(* IEC 61131-3 sources: Std_PalletMover/Class/MQTTClient_Interface (part 3) *)

      //-------------------------------
      //Logging
      //-------------------------------
      t_e_XML_Config::XC_Logging:

        if ProcessXML_ProcessConfig_Logging(pElement:=pThisElement) = FALSE then
          //CreateLog: Processing Logging Section of Configuration XML File Failed.

          Logging_InterfLog(usLevel     :=  MQTTCLIENTINTERFACE_LOGGING_LEVEL_ERR,
                            dMsgGroup   :=  MQCLIINF_LOG_ERROR_XML_CONFIG_LOGGING_NOT_OK_GRP,
                            dMsgNbr     :=  MQCLIINF_LOG_ERROR_XML_CONFIG_LOGGING_NOT_OK_MSG,
                            pMsg        :=  MQCLIINF_LOG_ERROR_XML_CONFIG_LOGGING_NOT_OK_TEXT,
                            pPara1      :=  NIL,
                            pPara2      :=  NIL,
                            pPara3      :=  NIL,
                            pPara4      :=  NIL);

          bOK := FALSE;
        end_if;

      //-------------------------------
      //Unknown, Skip
      //-------------------------------
      t_e_XML_Config::XC_Unknown:

    end_case;

    //Get the next client
    pThisElement := pThisElement^.pNext;

  end_while;

END_FUNCTION

FUNCTION MQTTClient_Interface::ProcessXML_ProcessConfig_GetElementType
	VAR_INPUT
		pElement 	: ^_XML_ELEMENT;
	END_VAR
	VAR_OUTPUT
		ElementType 	: t_e_XML_Config;
	END_VAR
  VAR
  	aString : ARRAY[0..MQTTCLIENT_INT_XML_CONFIG_MAX_LEN] of CHAR;
  END_VAR

  //Assume Unknown
  ElementType := XC_Unknown;

  if  pElement = NIL        |
      pElement^.Name = NIL  then
    return;
  end_if;

  //Convert the String to all upper for comparison to eliminate casing constraints
  SigCLib.StrNCpy(dst0  :=  #aString[0],
                  src0  :=  pElement^.Name,
                  count :=  MQTTCLIENT_INT_XML_CONFIG_MAX_LEN-1);

  aString[SigCLib.StrLen(str:=pElement^.Name)] := 0x00;

  SigCLib.StrUpr(ps1:=#aString[0]);

  if SigCLib.StrCmp(ps1:=#aString[0], ps2:=MQTTCLIENT_INT_XML_CONFIG_CLIENTID) = 0 then
    ElementType := XC_ClientID;
  elsif SigCLib.StrCmp(ps1:=#aString[0], ps2:=MQTTCLIENT_INT_XML_CONFIG_CONNECTION) = 0 then
    ElementType := XC_Connection;
  elsif SigCLib.StrCmp(ps1:=#aString[0], ps2:=MQTTCLIENT_INT_XML_CONFIG_RECONNECTION) = 0 then
    ElementType := XC_Reconnection;
  elsif SigCLib.StrCmp(ps1:=#aString[0], ps2:=MQTTCLIENT_INT_XML_CONFIG_TLS) = 0 then
    ElementType := XC_TLS;
  elsif SigCLib.StrCmp(ps1:=#aString[0], ps2:=MQTTCLIENT_INT_XML_CONFIG_LOGGING) = 0 then
    ElementType := XC_Logging;
  elsif SigCLib.StrCmp(ps1:=#aString[0], ps2:=MQTTCLIENT_INT_XML_CONFIG_WILL) = 0 then
    ElementType := XC_Will;
  end_if;

END_FUNCTION

FUNCTION MQTTClient_Interface::ProcessXML_ProcessConfig_ClientID
	VAR_INPUT
		pElement 	: ^_XML_ELEMENT;
	END_VAR
	VAR_OUTPUT
		bOK 	: BOOL;
	END_VAR

  //Assume Fail
  MQTTClientConfigData.Config.bClientIDSet := bOK := FALSE;

  //Get the ClientID from the XML File
  if  pElement                                                                              &
      pElement^.pText                                                                       &
      SigCLib.StrLen(str:=pElement^.pText) < sizeof(MQTTClientConfigData.Config.aClientID)  then

    SigCLib.MemSet( dst   :=  #MQTTClientConfigData.Config.aClientID[0],
                    c     :=  0x00,
                    len   :=  sizeof(MQTTClientConfigData.Config.aClientID));
    SigCLib.Utf8ToStr16(dst :=  #MQTTClientConfigData.Config.aClientID[0],
                        src :=  pElement^.pText);

    MQTTClientConfigData.Config.bClientIDSet := bOK := TRUE;

  end_if;

END_FUNCTION

FUNCTION MQTTClient_Interface::ProcessXML_GetElementType
	VAR_INPUT
		pElement 	: ^_XML_ELEMENT;
	END_VAR
	VAR_OUTPUT
		ElementType 	: t_e_XML;
	END_VAR
  VAR
  	aString : ARRAY[0..MTTCLIENT_INT_XML_CONFIG_DATAMAP_MAX_LEN] of CHAR;
  END_VAR

  //Assume Not Found
  ElementType := X_Unknown;

    //Convert the String to all upper for comparison to eliminate casing constraints
    SigCLib.StrNCpy(dst0  :=  #aString[0],
                    src0  :=  pElement^.Name,
                    count :=  MTTCLIENT_INT_XML_CONFIG_DATAMAP_MAX_LEN-1);

    aString[SigCLib.StrLen(str:=pElement^.Name)] := 0x00;

    SigCLib.StrUpr(ps1:=#aString[0]);

  if pElement then

    if SigCLib.StrCmp(ps1:=#aString[0], ps2:=MTTCLIENT_INT_XML_CONFIG_ELEMENT) = 0 then
      ElementType := X_Config;
      return;
    elsif SigCLib.StrCmp(ps1:=#aString[0], ps2:=MTTCLIENT_INT_XML_DATAMAP_ELEMENT) = 0 then
      ElementType := X_DataMap;
      return;
    end_if;

  end_if;

END_FUNCTION

FUNCTION MQTTClient_Interface::ProcessXML_ProcessDataMap
	VAR_INPUT
		pElement 	: ^_XML_ELEMENT;
	END_VAR
	VAR_OUTPUT
		bOK 	: BOOL;
	END_VAR
  VAR
  	pThisElement : ^_XML_ELEMENT;
  END_VAR

  //Assume Fail
  bOK := FALSE;

  if pElement = NIL then
    return;
  end_if;

  bOK := TRUE;
  pThisElement := pElement;

  //Step through all the children
  while pThisElement do

    //======================================================================
    //Based on the type of element, process
    //======================================================================
    case ProcessXML_ProcessDataMap_GetElementType(pElement:=pThisElement) of

      //-------------------------------
      //Unknown
      //-------------------------------
      t_e_XML_DataMap::XD_Unknown:

        //Create Log: Unexpected input in DataMap section

        Logging_InterfLog(usLevel     :=  MQTTCLIENTINTERFACE_LOGGING_LEVEL_ERR,
                          dMsgGroup   :=  MQCLIINF_LOG_ERROR_XML_DATAMAP_UNEXPECTED_ENTRY_GRP,
                          dMsgNbr     :=  MQCLIINF_LOG_ERROR_XML_DATAMAP_UNEXPECTED_ENTRY_MSG,
                          pMsg        :=  MQCLIINF_LOG_ERROR_XML_DATAMAP_UNEXPECTED_ENTRY_TEXT,
                          pPara1      :=  NIL,
                          pPara2      :=  NIL,
                          pPara3      :=  NIL,
                          pPara4      :=  NIL);

        bOK := FALSE;

      //-------------------------------
      //Topic Section
      //-------------------------------
      t_e_XML_DataMap::XD_TopicSection:

        if ProcessXML_ProcessDataMap_TopicSection(pElement:=pThisElement) = FALSE then

          bOK := FALSE;
          //Create Log: Failed Processing TopicSection in the DataMap Section

          Logging_InterfLog(usLevel     :=  MQTTCLIENTINTERFACE_LOGGING_LEVEL_ERR,
                            dMsgGroup   :=  MQCLIINF_LOG_ERROR_XML_DATAMAP_TOPICSECT_NOT_OK_GRP,
                            dMsgNbr     :=  MQCLIINF_LOG_ERROR_XML_DATAMAP_TOPICSECT_NOT_OK_MSG,
                            pMsg        :=  MQCLIINF_LOG_ERROR_XML_DATAMAP_TOPICSECT_NOT_OK_TEXT,
                            pPara1      :=  NIL,
                            pPara2      :=  NIL,
                            pPara3      :=  NIL,
                            pPara4      :=  NIL);
        end_if;

      //-------------------------------
      //Topic Endpoint
      //-------------------------------
      t_e_XML_DataMap::XD_TopicEndpoint:

        if ProcessXML_ProcessDataMap_TopicEndpoint(pElement:=pThisElement) = FALSE then
          bOK := FALSE;
          //Create Log: Failed Processing TopicEndpoint in the DataMap Section

          Logging_InterfLog(usLevel     :=  MQTTCLIENTINTERFACE_LOGGING_LEVEL_ERR,
                            dMsgGroup   :=  MQCLIINF_LOG_ERROR_XML_DATAMAP_TOPICENDPT_NOT_OK_GRP,
                            dMsgNbr     :=  MQCLIINF_LOG_ERROR_XML_DATAMAP_TOPICENDPT_NOT_OK_MSG,
                            pMsg        :=  MQCLIINF_LOG_ERROR_XML_DATAMAP_TOPICENDPT_NOT_OK_TEXT,
                            pPara1      :=  NIL,
                            pPara2      :=  NIL,
                            pPara3      :=  NIL,
                            pPara4      :=  NIL);

        end_if;

    end_case;

    pThisElement := pThisElement^.pNext;

  end_while;

END_FUNCTION

FUNCTION MQTTClient_Interface::ProcessXML_ProcessConfig_Connection
	VAR_INPUT
		pElement 	: ^_XML_ELEMENT;
	END_VAR
	VAR_OUTPUT
		bOK 	: BOOL;
	END_VAR
  VAR
    pThisElement : ^_XML_ELEMENT;
    aString : ARRAY[0..MQTTCLIENT_INT_XML_CONFIG_CONN_MAX_LEN] of CHAR;
  END_VAR

  bOK := FALSE;

  //Process the Connect Config
  if pElement             &
     pElement^.pChildren  then

    //==========================================================
    //Set Parameters
    //==========================================================
    pThisElement := pElement^.pChildren;

    while pThisElement        &
          pThisElement^.Name  &
          pThisElement^.pText do

      //Convert the String to all upper for comparison to eliminate casing constraints
      SigCLib.StrNCpy(dst0  :=  #aString[0],
                      src0  :=  pThisElement^.Name,
                      count :=  MQTTCLIENT_INT_XML_CONFIG_CONN_MAX_LEN-1);

      aString[SigCLib.StrLen(str:=pThisElement^.Name)] := 0x00;

      SigCLib.StrUpr(ps1:=#aString[0]);

      //------------------------------------------------------------------------------------------------------
      //Hostname
      //------------------------------------------------------------------------------------------------------
      if SigCLib.StrCmp(ps1:=#aString[0], ps2:=MQTTCLIENT_INT_XML_CONFIG_CONN_HOSTNAME) = 0 then

        if SigCLib.StrLen(str:=pThisElement^.pText) < MQTTCLIENT_HOSTNAME_MAX_LEN then
          SigCLib.Utf8ToStr16(dst:=#MQTTClientConfigData.Config.Connect.aHostname[0], src:=pThisElement^.pText);
          MQTTClientConfigData.Config.Connect.ValuesSet.Hostname := TRUE;
        end_if;

      //------------------------------------------------------------------------------------------------------
      //Port
      //------------------------------------------------------------------------------------------------------
      elsif SigCLib.StrCmp(ps1:=#aString[0], ps2:=MQTTCLIENT_INT_XML_CONFIG_CONN_PORT) = 0 then

        if SigCLib.StrLen(str:=pThisElement^.pText) < MQTTCLIENTINTERFACE_CONNECT_PORT_MAX_LEN then
          MQTTClientConfigData.Config.Connect.iPort := to_int(SigCLib.AToI(ps1:=pThisElement^.pText));
          MQTTClientConfigData.Config.Connect.ValuesSet.Port := TRUE;
        end_if;

      //------------------------------------------------------------------------------------------------------
      //Keepalive
      //------------------------------------------------------------------------------------------------------
      elsif SigCLib.StrCmp(ps1:=#aString[0], ps2:=MQTTCLIENT_INT_XML_CONFIG_CONN_KEEPALIVE) = 0 then

        if SigCLib.StrLen(str:=pThisElement^.pText) < MQTTCLIENTINTERFACE_CONNECT_KEEPALIVE_MAX_LEN then
          MQTTClientConfigData.Config.Connect.iKeepalive := to_int(SigCLib.AToI(ps1:=pThisElement^.pText));
          MQTTClientConfigData.Config.Connect.ValuesSet.Keepalive := TRUE;
        end_if;

      //------------------------------------------------------------------------------------------------------
      //Max Inflight
      //------------------------------------------------------------------------------------------------------
      elsif SigCLib.StrCmp(ps1:=#aString[0], ps2:=MQTTCLIENT_INT_XML_CONFIG_CONN_MAXINFLIGHT) = 0 then

        if SigCLib.StrLen(str:=pThisElement^.pText) < MQTTCLIENTINTERFACE_CONNECT_INFLIGHT_MAX_LEN then
          MQTTClientConfigData.Config.Connect.iMaxInflightMessages := to_int(SigCLib.AToI(ps1:=pThisElement^.pText));
          MQTTClientConfigData.Config.Connect.ValuesSet.MaxInflight := TRUE;
        end_if;

      //------------------------------------------------------------------------------------------------------
      //Username
      //------------------------------------------------------------------------------------------------------
      elsif SigCLib.StrCmp(ps1:=#aString[0], ps2:=MQTTCLIENT_INT_XML_CONFIG_CONN_USERNAME) = 0 then

        if SigCLib.StrLen(str:=pThisElement^.pText) < MQTTCLIENTINTERFACE_CONNECT_USERNAME_MAX_LEN then
          SigCLib.Utf8ToStr16(dst:=#MQTTClientConfigData.Config.Connect.aUsername[0], src:=pThisElement^.pText);
          MQTTClientConfigData.Config.Connect.ValuesSet.Username := TRUE;
        end_if;

      //------------------------------------------------------------------------------------------------------
      //Password
      //------------------------------------------------------------------------------------------------------
      elsif SigCLib.StrCmp(ps1:=#aString[0], ps2:=MQTTCLIENT_INT_XML_CONFIG_CONN_PASSWORD) = 0 then

        if SigCLib.StrLen(str:=pThisElement^.pText) < MQTTCLIENTINTERFACE_CONNECT_PASSWORD_MAX_LEN then
          SigCLib.Utf8ToStr16(dst:=#MQTTClientConfigData.Config.Connect.aPassword[0], src:=pThisElement^.pText);
          MQTTClientConfigData.Config.Connect.ValuesSet.Password := TRUE;
        end_if;

      end_if;

      pThisElement := pThisElement^.pNext;

    end_while;

    //Return is OK if atleast the Hostname is set
    bOK := MQTTClientConfigData.Config.Connect.ValuesSet.Hostname;

  end_if;

END_FUNCTION

FUNCTION MQTTClient_Interface::ProcessXML_ProcessConfig_Will
	VAR_INPUT
		pElement 	: ^_XML_ELEMENT;
	END_VAR
	VAR_OUTPUT
		bOK 	: BOOL;
	END_VAR
  VAR
    pThisElement : ^_XML_ELEMENT;
  	aString : ARRAY[0..MQTTCLIENT_INT_XML_CONFIG_WILL_MAX_LEN] of CHAR;
  END_VAR

  bOK := FALSE;

  //Process the Connect Config
  if pElement             &
     pElement^.pChildren  then

    //==========================================================
    //Set Parameters
    //==========================================================
    pThisElement := pElement^.pChildren;

    while pThisElement        &
          pThisElement^.Name  &
          pThisElement^.pText do

      //Convert the String to all upper for comparison to eliminate casing constraints
      SigCLib.StrNCpy(dst0  :=  #aString[0],
                      src0  :=  pThisElement^.Name,
                      count :=  MQTTCLIENT_INT_XML_CONFIG_WILL_MAX_LEN-1);

      aString[SigCLib.StrLen(str:=pThisElement^.Name)] := 0x00;

      SigCLib.StrUpr(ps1:=#aString[0]);

      //------------------------------------------------------------------------------------------------------
      //Topic
      //------------------------------------------------------------------------------------------------------
      if SigCLib.StrCmp(ps1:=#aString[0], ps2:=MQTTCLIENT_INT_XML_CONFIG_WILL_TOPIC) = 0 then

        if SigCLib.StrLen(str:=pThisElement^.pText) < MQTTCLIENTINTERFACE_WILL_TOPIC_MAX_LEN then
          SigCLib.Utf8ToStr16(dst:=#MQTTClientConfigData.Config.Will.aTopic[0], src:=pThisElement^.pText);
          MQTTClientConfigData.Config.Will.ValuesSet.Topic := TRUE;
        end_if;

      //------------------------------------------------------------------------------------------------------
      //Payload
      //------------------------------------------------------------------------------------------------------
      elsif SigCLib.StrCmp(ps1:=#aString[0], ps2:=MQTTCLIENT_INT_XML_CONFIG_WILL_PLTEXT) = 0 then

        if SigCLib.StrLen(str:=pThisElement^.pText) < MQTTCLIENTINTERFACE_WILL_PAYLOAD_MAX_LEN then
          //Data from XML Structure must be text, although the payload in the MQTT Client allows for Non-UTF8 input
          SigCLib.StrCpy(dst0:=#MQTTClientConfigData.Config.Will.aPayload[0], src0:=pThisElement^.pText);
          MQTTClientConfigData.Config.Will.ValuesSet.Payload := TRUE;
        end_if;

      //------------------------------------------------------------------------------------------------------
      //QoS
      //------------------------------------------------------------------------------------------------------
      elsif SigCLib.StrCmp(ps1:=#aString[0], ps2:=MQTTCLIENT_INT_XML_CONFIG_WILL_QOS) = 0 then

        if SigCLib.StrLen(str:=pThisElement^.pText) = MQTTCLIENTINTERFACE_WILL_QOS_MAX_LEN then

          MQTTClientConfigData.Config.Will.ValuesSet.QoS := TRUE;

          //=======================================
          //Conv QoS CHAR to INT
          //=======================================
          case pThisElement^.pText^ of
            //-----------------------------------
            //QoS 0
            //-----------------------------------
            MQTTCLIENT_INT_XML_CONFIG_WILL_QOS_0:

              MQTTClientConfigData.Config.Will.iQoS := 0;

            //-----------------------------------
            //QoS 1
            //-----------------------------------
            MQTTCLIENT_INT_XML_CONFIG_WILL_QOS_1:

              MQTTClientConfigData.Config.Will.iQoS := 1;

            //-----------------------------------
            //QoS 2
            //-----------------------------------
            MQTTCLIENT_INT_XML_CONFIG_WILL_QOS_2:

              MQTTClientConfigData.Config.Will.iQoS := 2;

          //Not a valid Character
          else

            MQTTClientConfigData.Config.Will.ValuesSet.QoS := FALSE;

          end_case;

        end_if;

      //------------------------------------------------------------------------------------------------------
      //Retain
      //------------------------------------------------------------------------------------------------------
      elsif SigCLib.StrCmp(ps1:=#aString[0], ps2:=MQTTCLIENT_INT_XML_CONFIG_WILL_RETAIN) = 0 then

        if SigCLib.StrLen(str:=pThisElement^.pText) = MQTTCLIENT_INT_XML_CONFIG_WILL_RETAIN_MAXLEN then

          //===========================
          //Set Log based on text value
          //===========================
          case pThisElement^.pText^ of
            //---------------------------------
            //True
            //---------------------------------
            MQTTCLIENT_INT_XML_CONFIG_WILL_RETAIN_TRUE:
              MQTTClientConfigData.Config.Will.bRetain := TRUE;
              MQTTClientConfigData.Config.Will.ValuesSet.RetainWill := TRUE;
            //---------------------------------
            //False
            //---------------------------------
            MQTTCLIENT_INT_XML_CONFIG_WILL_RETAIN_FALSE:
              MQTTClientConfigData.Config.Will.bRetain := FALSE;
              MQTTClientConfigData.Config.Will.ValuesSet.RetainWill := TRUE;
          end_case;

        end_if;

      end_if;

      pThisElement := pThisElement^.pNext;

    end_while;

    //All Paras are required
    bOK :=  MQTTClientConfigData.Config.Will.ValuesSet.Topic      &
            MQTTClientConfigData.Config.Will.ValuesSet.Payload    &
            MQTTClientConfigData.Config.Will.ValuesSet.QoS        &
            MQTTClientConfigData.Config.Will.ValuesSet.RetainWill;

  end_if;

END_FUNCTION

FUNCTION MQTTClient_Interface::ProcessXML_ProcessConfig_Reconnection
	VAR_INPUT
		pElement 	: ^_XML_ELEMENT;
	END_VAR
	VAR_OUTPUT
		bOK 	: BOOL;
	END_VAR
  VAR
    pThisElement : ^_XML_ELEMENT;
    aString : ARRAY[0..MQTTCLIENT_INT_XML_CONFIG_RECONN_MAXLEN] of CHAR;
  END_VAR

  bOK := FALSE;

  //Process the Connect Config
  if pElement             &
     pElement^.pChildren  then

    //==========================================================
    //Set Parameters
    //==========================================================
    pThisElement := pElement^.pChildren;

    while pThisElement        &
          pThisElement^.Name  &
          pThisElement^.pText do

      //Convert the String to all upper for comparison to eliminate casing constraints
      SigCLib.StrNCpy(dst0  :=  #aString[0],
                      src0  :=  pThisElement^.Name,
                      count :=  MQTTCLIENT_INT_XML_CONFIG_RECONN_MAXLEN-1);

      aString[SigCLib.StrLen(str:=pThisElement^.Name)] := 0x00;

      SigCLib.StrUpr(ps1:=#aString[0]);

      //------------------------------------------------------------------------------------------------------
      //Min Interval
      //------------------------------------------------------------------------------------------------------
      if SigCLib.StrCmp(ps1:=#aString[0], ps2:=MQTTCLIENT_INT_XML_CONFIG_RECONN_MININT) = 0 then

        if SigCLib.StrLen(str:=pThisElement^.pText) < MQTTCLIENTINTERFACE_RECONNECT_MININT_MAX_LEN then
          MQTTClientConfigData.Config.Reconnect.iMinInterval := to_int(SigCLib.AToI(ps1:=pThisElement^.pText));
          MQTTClientConfigData.Config.Reconnect.ValuesSet.MinInterval := TRUE;
        end_if;

      //------------------------------------------------------------------------------------------------------
      //Max Interval
      //------------------------------------------------------------------------------------------------------
      elsif SigCLib.StrCmp(ps1:=#aString[0], ps2:=MQTTCLIENT_INT_XML_CONFIG_RECONN_MAXINT) = 0 then

        if SigCLib.StrLen(str:=pThisElement^.pText) < MQTTCLIENTINTERFACE_RECONNECT_MAXINT_MAX_LEN then
          MQTTClientConfigData.Config.Reconnect.iMaxInterval := to_int(SigCLib.AToI(ps1:=pThisElement^.pText));
          MQTTClientConfigData.Config.Reconnect.ValuesSet.MaxInterval := TRUE;
        end_if;

      //------------------------------------------------------------------------------------------------------
      //Exponential Scale
      //------------------------------------------------------------------------------------------------------
      elsif SigCLib.StrCmp(ps1:=#aString[0], ps2:=MQTTCLIENT_INT_XML_CONFIG_RECONN_EXPSCALE) = 0 then

        if SigCLib.StrLen(str:=pThisElement^.pText) = SigCLib.StrLen(str:=MQTTCLIENT_INT_XML_CONFIG_RECONNECT_EXP_ON) then
          MQTTClientConfigData.Config.Reconnect.bExponential := (SigCLib.StrCmp(ps1:=pThisElement^.pText, ps2:=MQTTCLIENT_INT_XML_CONFIG_RECONNECT_EXP_ON) = 0);
          MQTTClientConfigData.Config.Reconnect.ValuesSet.ExponentialScale := TRUE;
        end_if;

      end_if;

      pThisElement := pThisElement^.pNext;

    end_while;

    //Return is OK if all is set
    bOK :=  MQTTClientConfigData.Config.Reconnect.ValuesSet.MinInterval &
            MQTTClientConfigData.Config.Reconnect.ValuesSet.MaxInterval &
            MQTTClientConfigData.Config.Reconnect.ValuesSet.ExponentialScale;

  end_if;

END_FUNCTION

FUNCTION MQTTClient_Interface::ProcessXML_ProcessConfig_TLS
	VAR_INPUT
		pElement 	: ^_XML_ELEMENT;
	END_VAR
	VAR_OUTPUT
		bOK 	: BOOL;
	END_VAR
  VAR
    pThisElement : ^_XML_ELEMENT;
    aString : ARRAY[0..MQTTCLIENT_INT_XML_CONFIG_TLS_MAXLEN] of CHAR;
  END_VAR

  bOK := FALSE;

  //Process the Connect Config
  if pElement             &
     pElement^.pChildren  then

    MQTTClientConfigData.Config.TLS.ValuesSet.TLS := TRUE;

    //==========================================================
    //Set Parameters
    //==========================================================
    pThisElement := pElement^.pChildren;

    while pThisElement        &
          pThisElement^.Name  &
          pThisElement^.pText do

      //Convert the String to all upper for comparison to eliminate casing constraints
      SigCLib.StrNCpy(dst0  :=  #aString[0],
                      src0  :=  pThisElement^.Name,
                      count :=  MQTTCLIENT_INT_XML_CONFIG_TLS_MAXLEN-1);

      aString[SigCLib.StrLen(str:=pThisElement^.Name)] := 0x00;

      SigCLib.StrUpr(ps1:=#aString[0]);

      //------------------------------------------------------------------------------------------------------
      //cafile
      //------------------------------------------------------------------------------------------------------
      if SigCLib.StrCmp(ps1:=#aString[0], ps2:=MQTTCLIENT_INT_XML_CONFIG_TLS_CAFILE) = 0 then

        if SigCLib.StrLen(str:=pThisElement^.pText) < MQTTCLIENTINTERFACE_TLS_CAFILE_MAX_LEN then
          SigCLib.StrCpy(dst0:=#MQTTClientConfigData.Config.TLS.aCAFile[0], src0:=pThisElement^.pText);
          MQTTClientConfigData.Config.TLS.ValuesSet.CAFile := TRUE;
        end_if;

      //------------------------------------------------------------------------------------------------------
      //certfile
      //------------------------------------------------------------------------------------------------------
      elsif SigCLib.StrCmp(ps1:=#aString[0], ps2:=MQTTCLIENT_INT_XML_CONFIG_TLS_CERTFILE) = 0 then

        if SigCLib.StrLen(str:=pThisElement^.pText) < MQTTCLIENTINTERFACE_TLS_CERTFILE_MAX_LEN then
          SigCLib.StrCpy(dst0:=#MQTTClientConfigData.Config.TLS.aCertFile[0], src0:=pThisElement^.pText);
          MQTTClientConfigData.Config.TLS.ValuesSet.CertFile := TRUE;
        end_if;

      //------------------------------------------------------------------------------------------------------
      //keyfile
      //------------------------------------------------------------------------------------------------------
      elsif SigCLib.StrCmp(ps1:=#aString[0], ps2:=MQTTCLIENT_INT_XML_CONFIG_TLS_KEYFILE) = 0 then

        if SigCLib.StrLen(str:=pThisElement^.pText) < MQTTCLIENTINTERFACE_TLS_KEYFILE_MAX_LEN then
          SigCLib.StrCpy(dst0:=#MQTTClientConfigData.Config.TLS.aKeyFile[0], src0:=pThisElement^.pText);
          MQTTClientConfigData.Config.TLS.ValuesSet.KeyFile := TRUE;
        end_if;

      //------------------------------------------------------------------------------------------------------
      //pw
      //------------------------------------------------------------------------------------------------------
      elsif SigCLib.StrCmp(ps1:=#aString[0], ps2:=MQTTCLIENT_INT_XML_CONFIG_TLS_PW) = 0 then

        if SigCLib.StrLen(str:=pThisElement^.pText) < MQTTCLIENTINTERFACE_TLS_PASSWORD_MAX_LEN then
          SigCLib.StrCpy(dst0:=#MQTTClientConfigData.Config.TLS.aPassword[0], src0:=pThisElement^.pText);
          MQTTClientConfigData.Config.TLS.ValuesSet.Password := TRUE;
        end_if;

      end_if;

      pThisElement := pThisElement^.pNext;

    end_while;

    //No input is required
    bOK := TRUE;

  end_if;

END_FUNCTION

FUNCTION MQTTClient_Interface::ProcessXML_ProcessConfig_Logging
	VAR_INPUT
		pElement 	: ^_XML_ELEMENT;
	END_VAR
	VAR_OUTPUT
		bOK 	: BOOL;
	END_VAR
  VAR
    pThisElement : ^_XML_ELEMENT;
    aString : ARRAY[0..MQTTCLIENT_INT_XML_CONFIG_LOG_MAX_LEN] of CHAR;
  END_VAR

  bOK := FALSE;

  MQTTClientConfigData.Config.Logging.bLogSet       := FALSE;
  MQTTClientConfigData.Config.Logging.bdActiveLogs  := 0;

  //Process the Logging Config
  if pElement             &
     pElement^.pChildren  then

    //==========================================================
    //Set Parameters
    //==========================================================
    pThisElement := pElement^.pChildren;

    while pThisElement        &
          pThisElement^.Name  &
          pThisElement^.pText do

      //Convert the String to all upper for comparison to eliminate casing constraints
      SigCLib.StrNCpy(dst0  :=  #aString[0],
                      src0  :=  pThisElement^.Name,
                      count :=  MQTTCLIENT_INT_XML_CONFIG_LOG_MAX_LEN-1);

      aString[SigCLib.StrLen(str:=pThisElement^.Name)] := 0x00;

      SigCLib.StrUpr(ps1:=#aString[0]);

      //If any log entry is present, set the ValuePresent
      MQTTClientConfigData.Config.Logging.bLogSet := TRUE;

      //------------------------------------------------------------------------------------------------------
      //Info
      //------------------------------------------------------------------------------------------------------
      if SigCLib.StrCmp(ps1:=#aString[0], ps2:=MQTTCLIENT_INT_XML_CONFIG_LOG_INFO) = 0 then

        if SigCLib.StrLen(str:=pThisElement^.pText) = MQTTCLIENTINTERFACE_LOG_ON_OFF_MAX_LEN then

          //===========================
          //Set Log based on text value
          //===========================
          case pThisElement^.pText^ of
            //---------------------------------
            //Off
            //---------------------------------
            MQTTCLIENT_INT_XML_CONFIG_LOG_OFF:
              MQTTClientConfigData.Config.Logging.bdActiveLogs$BDINT := MQTTClientConfigData.Config.Logging.bdActiveLogs$BDINT AND (NOT (MQTTCLIENTINTERFACE_LOGGING_LEVEL_INFO$BDINT));
            //---------------------------------
            //On
            //---------------------------------
            MQTTCLIENT_INT_XML_CONFIG_LOG_ON:
              MQTTClientConfigData.Config.Logging.bdActiveLogs$BDINT := MQTTClientConfigData.Config.Logging.bdActiveLogs$BDINT OR MQTTCLIENTINTERFACE_LOGGING_LEVEL_INFO$BDINT;
          end_case;

        end_if;

      //------------------------------------------------------------------------------------------------------
      //Notice
      //------------------------------------------------------------------------------------------------------
      elsif SigCLib.StrCmp(ps1:=#aString[0], ps2:=MQTTCLIENT_INT_XML_CONFIG_LOG_NOTICE) = 0 then

        if SigCLib.StrLen(str:=pThisElement^.pText) = MQTTCLIENTINTERFACE_LOG_ON_OFF_MAX_LEN then

          //===========================
          //Set Log based on text value
          //===========================
          case pThisElement^.pText^ of
            //---------------------------------
            //Off
            //---------------------------------
            MQTTCLIENT_INT_XML_CONFIG_LOG_OFF:
              MQTTClientConfigData.Config.Logging.bdActiveLogs$BDINT := MQTTClientConfigData.Config.Logging.bdActiveLogs$BDINT AND (NOT (MQTTCLIENTINTERFACE_LOGGING_LEVEL_NOTICE$BDINT));
            //---------------------------------
            //On
            //---------------------------------
            MQTTCLIENT_INT_XML_CONFIG_LOG_ON:
              MQTTClientConfigData.Config.Logging.bdActiveLogs := MQTTClientConfigData.Config.Logging.bdActiveLogs OR MQTTCLIENTINTERFACE_LOGGING_LEVEL_NOTICE$BDINT;
          end_case;

        end_if;

      //------------------------------------------------------------------------------------------------------
      //Warning
      //------------------------------------------------------------------------------------------------------
      elsif SigCLib.StrCmp(ps1:=#aString[0], ps2:=MQTTCLIENT_INT_XML_CONFIG_LOG_WARNING) = 0 then

        if SigCLib.StrLen(str:=pThisElement^.pText) = MQTTCLIENTINTERFACE_LOG_ON_OFF_MAX_LEN then

          //===========================
          //Set Log based on text value
          //===========================
          case pThisElement^.pText^ of
            //---------------------------------
            //Off
            //---------------------------------
            MQTTCLIENT_INT_XML_CONFIG_LOG_OFF:
              MQTTClientConfigData.Config.Logging.bdActiveLogs$BDINT := MQTTClientConfigData.Config.Logging.bdActiveLogs$BDINT AND (NOT MQTTCLIENTINTERFACE_LOGGING_LEVEL_WARNING);
            //---------------------------------
            //On
            //---------------------------------
            MQTTCLIENT_INT_XML_CONFIG_LOG_ON:
              MQTTClientConfigData.Config.Logging.bdActiveLogs := MQTTClientConfigData.Config.Logging.bdActiveLogs OR MQTTCLIENTINTERFACE_LOGGING_LEVEL_WARNING$BDINT;
          end_case;

        end_if;

      //------------------------------------------------------------------------------------------------------
      //Error
      //------------------------------------------------------------------------------------------------------
      elsif SigCLib.StrCmp(ps1:=#aString[0], ps2:=MQTTCLIENT_INT_XML_CONFIG_LOG_ERROR) = 0 then

        if SigCLib.StrLen(str:=pThisElement^.pText) = MQTTCLIENTINTERFACE_LOG_ON_OFF_MAX_LEN then

          //===========================
          //Set Log based on text value
          //===========================
          case pThisElement^.pText^ of
            //---------------------------------
            //Off
            //---------------------------------
            MQTTCLIENT_INT_XML_CONFIG_LOG_OFF:
              MQTTClientConfigData.Config.Logging.bdActiveLogs$BDINT := MQTTClientConfigData.Config.Logging.bdActiveLogs$BDINT AND (NOT (MQTTCLIENTINTERFACE_LOGGING_LEVEL_ERR$BDINT));
            //---------------------------------
            //On
            //---------------------------------
            MQTTCLIENT_INT_XML_CONFIG_LOG_ON:
              MQTTClientConfigData.Config.Logging.bdActiveLogs$BDINT := MQTTClientConfigData.Config.Logging.bdActiveLogs$BDINT OR MQTTCLIENTINTERFACE_LOGGING_LEVEL_ERR$BDINT;
          end_case;

        end_if;

      //------------------------------------------------------------------------------------------------------
      //Debugging
      //------------------------------------------------------------------------------------------------------
      elsif SigCLib.StrCmp(ps1:=#aString[0], ps2:=MQTTCLIENT_INT_XML_CONFIG_LOG_DEBUGGING) = 0 then

        if SigCLib.StrLen(str:=pThisElement^.pText) = MQTTCLIENTINTERFACE_LOG_ON_OFF_MAX_LEN then

          //===========================
          //Set Log based on text value
          //===========================
          case pThisElement^.pText^ of
            //---------------------------------
            //Off
            //---------------------------------
            MQTTCLIENT_INT_XML_CONFIG_LOG_OFF:
              MQTTClientConfigData.Config.Logging.bdActiveLogs$BDINT := MQTTClientConfigData.Config.Logging.bdActiveLogs$BDINT AND (NOT (MQTTCLIENTINTERFACE_LOGGING_LEVEL_DEBUG$BDINT));
            //---------------------------------
            //On
            //---------------------------------
            MQTTCLIENT_INT_XML_CONFIG_LOG_ON:
              MQTTClientConfigData.Config.Logging.bdActiveLogs$BDINT := MQTTClientConfigData.Config.Logging.bdActiveLogs$BDINT OR MQTTCLIENTINTERFACE_LOGGING_LEVEL_DEBUG$BDINT;
          end_case;

        end_if;

      end_if;

      pThisElement := pThisElement^.pNext;

    end_while;

    //Return is always OK
    bOK := TRUE;

  end_if;

END_FUNCTION

FUNCTION MQTTClient_Interface::ProcessXML_ProcessDataMap_GetElementType
	VAR_INPUT
		pElement 	: ^_XML_ELEMENT;
	END_VAR
	VAR_OUTPUT
		ElementType 	: t_e_XML_DataMap;
	END_VAR
  VAR
  	aString : ARRAY[0..MQTTCLIENT_INT_XML_DATAMAP_TOPIC_SECT_END_MAX_LEN] of CHAR;
  END_VAR

  //Assume Unknown
  ElementType := XD_Unknown;

  if pElement then

  //Convert the String to all upper for comparison to eliminate casing constraints
    SigCLib.StrNCpy(dst0  :=  #aString[0],
                    src0  :=  pElement^.Name,
                    count :=  MQTTCLIENT_INT_XML_DATAMAP_TOPIC_SECT_END_MAX_LEN-1);

    aString[SigCLib.StrLen(str:=pElement^.Name)] := 0x00;

    SigCLib.StrUpr(ps1:=#aString[0]);

    if SigCLib.StrCmp(ps1:=#aString[0], ps2:=MQTTCLIENT_INT_XML_DATAMAP_TOPICSECTION) = 0 then
      ElementType := XD_TopicSection;
    elsif SigCLib.StrCmp(ps1:=#aString[0], ps2:=MQTTCLIENT_INT_XML_DATAMAP_TOPICENDPOINT) = 0 then
      ElementType := XD_TopicEndpoint;
    end_if;

  end_if;

END_FUNCTION

FUNCTION MQTTClient_Interface::ProcessXML_ProcessDataMap_TopicSection
	VAR_INPUT
		pElement 	: ^_XML_ELEMENT;
	END_VAR
	VAR_OUTPUT
		bOK 	: BOOL;
	END_VAR
  VAR
  	pChild : ^_XML_ELEMENT;
    tmpPara : DINT;
  	aString : ARRAY[0..MQTTCLIENT_INT_XML_DATAMAP_TOPICSECTION_ATTR_MAX_LEN] of CHAR;
  END_VAR

  //Assume Fail
  bOK := FALSE;

  if pElement = NIL                           |
     pElement^.Attributes.pList = NIL         |
     pElement^.Attributes.pList^.Name = NIL   |
     pElement^.Attributes.pList^.Value = NIL then
    return;
  end_if;

  //Convert the String to all upper for comparison to eliminate casing constraints
    SigCLib.StrNCpy(dst0  :=  #aString[0],
                    src0  :=  pElement^.Attributes.pList^.Name,
                    count :=  MQTTCLIENT_INT_XML_DATAMAP_TOPICSECTION_ATTR_MAX_LEN-1);

    aString[SigCLib.StrLen(str:=pElement^.Attributes.pList^.Name)] := 0x00;

    SigCLib.StrUpr(ps1:=#aString[0]);

  //Append the section to the Topicname being built (First and only Attribute should be "name")
  if SigCLib.StrCmp(ps1:=#aString[0], ps2:=MQTTCLIENT_INT_XML_DATAMAP_TOPICSECTION_ATTR_NAME) = 0 then

    //Topic Depth OK
    if Config.pDataMapConfig^.udTopicStringDepth >= 0 &
       Config.pDataMapConfig^.udTopicStringDepth <  MQTTCLIENT_INT_XML_DATAMAP_TOPICSECTION_MAXSECDEPTH then

      //Value set but too long
      if  (SigCLib.StrLen(str:=pElement^.Attributes.pList^.Value) >= MQTTCLIENT_INT_XML_DATAMAP_TOPICSECTION_MAXSECLEN) then

        //Create Log: DataMap, Processing topic Section failed - Section title too long

        Logging_InterfLog(usLevel     :=  MQTTCLIENTINTERFACE_LOGGING_LEVEL_ERR,
                          dMsgGroup   :=  MQCLIINF_LOG_ERROR_XML_DATAMAP_TS_TITLE_LEN_GRP,
                          dMsgNbr     :=  MQCLIINF_LOG_ERROR_XML_DATAMAP_TS_TITLE_LEN_MSG,
                          pMsg        :=  MQCLIINF_LOG_ERROR_XML_DATAMAP_TS_TITLE_LEN_TEXT,
                          pPara1      :=  NIL,
                          pPara2      :=  NIL,
                          pPara3      :=  NIL,
                          pPara4      :=  NIL);

        return;

      //Value not set
      elsif pElement^.Attributes.pList^.Value = NIL then

        //Create Log: DataMap, Processing topic Section failed - Section title empty

        Logging_InterfLog(usLevel     :=  MQTTCLIENTINTERFACE_LOGGING_LEVEL_ERR,
                          dMsgGroup   :=  MQCLIINF_LOG_ERROR_XML_DATAMAP_TS_TITLE_EMPTY_GRP,
                          dMsgNbr     :=  MQCLIINF_LOG_ERROR_XML_DATAMAP_TS_TITLE_EMPTY_MSG,
                          pMsg        :=  MQCLIINF_LOG_ERROR_XML_DATAMAP_TS_TITLE_EMPTY_TEXT,
                          pPara1      :=  NIL,
                          pPara2      :=  NIL,
                          pPara3      :=  NIL,
                          pPara4      :=  NIL);

        return;

      //Value set and OK
      else

        SigCLib.MemSet( dst :=  #Config.pDataMapConfig^.aTopicStrings[Config.pDataMapConfig^.udTopicStringDepth][0],
                        c   :=  0x00,
                        len :=  sizeof(t_s_TopicString));
        SigCLib.StrCpy( dst0  :=  #Config.pDataMapConfig^.aTopicStrings[Config.pDataMapConfig^.udTopicStringDepth][0],
                        src0  :=  pElement^.Attributes.pList^.Value);
        Config.pDataMapConfig^.udTopicStringDepth += 1;
        bOK := TRUE;

      end_if;

    //Exceeded maximum topic depth
    elsif Config.pDataMapConfig^.udTopicStringDepth >= MQTTCLIENT_INT_XML_DATAMAP_TOPICSECTION_MAXSECDEPTH then

      //Create Log: DataMap, Processing topic section failed, maximum topic depth exceeded.

      tmpPara := MQTTCLIENT_INT_XML_DATAMAP_TOPICSECTION_MAXSECDEPTH;

      Logging_InterfLog(usLevel     :=  MQTTCLIENTINTERFACE_LOGGING_LEVEL_ERR,
                        dMsgGroup   :=  MQCLIINF_LOG_ERROR_XML_DATAMAP_TS_MAX_DEPTH_EXCEED_GRP,
                        dMsgNbr     :=  MQCLIINF_LOG_ERROR_XML_DATAMAP_TS_MAX_DEPTH_EXCEED_MSG,
                        pMsg        :=  MQCLIINF_LOG_ERROR_XML_DATAMAP_TS_MAX_DEPTH_EXCEED_TEXT,
                        pPara1      :=  #Config.pDataMapConfig^.udTopicStringDepth$DINT,
                        pPara2      :=  #tmpPara,
                        pPara3      :=  NIL,
                        pPara4      :=  NIL);

    end_if;

    //Process any children the Section has
    pChild := pElement^.pChildren;
    if pChild then
      bOK := ProcessXML_ProcessDataMap(pElement:=pChild);
    else
      bOK := FALSE;
    end_if;

    if Config.pDataMapConfig^.udTopicStringDepth >= 1 then
      Config.pDataMapConfig^.udTopicStringDepth -= 1;
    end_if;

  end_if;

END_FUNCTION

FUNCTION MQTTClient_Interface::ProcessXML_ProcessDataMap_TopicEndpoint
	VAR_INPUT
		pElement 	: ^_XML_ELEMENT;
	END_VAR
	VAR_OUTPUT
		bOK 	: BOOL;
	END_VAR
  VAR
    aTopicString    : ARRAY[0..MQTTCLIENT_TOPIC_MAX_LEN] of CHAR;
  	udAtt, udCount  : UDINT;
    pAtt            : ^_XML_ATTRIBUTE;
    aEndpointName   : ARRAY[0..MQTTCLIENT_INT_XML_DATAMAP_TOPICENDPOINT_NAME_MAX_LEN] of CHAR;
    aElement        : ARRAY[0..MQTTCLIENT_INT_XML_DATAMAP_TOPICENDPOINT_ELEMENT_MAX_LEN] of CHAR;
    Operation       : t_e_DataMap_Operations;
    udInterval      : UDINT;
    DataType        : t_e_DataMap_DataTypes;
    bNameSet, bElementSet : BOOL;
    udLen           : UDINT;
    iQoS            : INT;
    DRSRetain       : t_e_DataMap_RetainStates;
    DataMapRet      : t_e_DataMap_RetCode;
    tmpPara         : DINT;
    aString         : ARRAY[0..MQTTCLIENT_INT_XML_DATAMAP_TOPICENDPOINT_ATTR_MAX_LEN] of CHAR;
  END_VAR

  //Assume Fail
  bOK := FALSE;

  if pElement = NIL                                                                 |
     pElement^.Attributes.no = 0                                                    |
     pElement^.Attributes.no > MQTTCLIENT_INT_XML_DATAMAP_TOPICENDPOINT_MAX_ATTRS   |
     pElement^.Attributes.pList = NIL                                               then
    return;
  end_if;

  //Set Default Values
  Operation   := DO_Subscribe;
  udInterval  := 0;
  DataType    := DD_DINT;
  bNameSet    := bElementSet := FALSE;
  iQoS        := 0;
  DRSRetain   := DRS_False;

  udAtt := pElement^.Attributes.no;

  while udAtt > 0 do

    //=======================
    //Process the Attribute
    //=======================
    pAtt := ((pElement^.Attributes.pList$UDINT) + (udAtt-1)*sizeof(_XML_ATTRIBUTE))$^_XML_ATTRIBUTE;

    if pAtt^.Name = NIL |
       pAtt^.Value = NIL then
      return;
    end_if;

    //Convert the String to all upper for comparison to eliminate casing constraints
    SigCLib.StrNCpy(dst0  :=  #aString[0],
                    src0  :=  pAtt^.Name$^CHAR,
                    count :=  MQTTCLIENT_INT_XML_DATAMAP_TOPICENDPOINT_ATTR_MAX_LEN-1);

    aString[SigCLib.StrLen(str:=pAtt^.Name$^CHAR)] := 0x00;

    SigCLib.StrUpr(ps1:=#aString[0]);

    //------------------------
    //Name
    //------------------------
    if SigCLib.StrCmp(ps1:=#aString[0], ps2:=MQTTCLIENT_INT_XML_DATAMAP_TOPICENDPOINT_ATTR_NAME) = 0 then

      udLen := SigCLib.StrLen(str:=pAtt^.Value$^CHAR);

      if udLen > MQTTCLIENT_INT_XML_DATAMAP_TOPICENDPOINT_NAME_MAX_LEN |
         udLen = 0                                                        then
        //Create Log: DataMap, Element text too long

        tmpPara := to_dint(udLen);

        Logging_InterfLog(usLevel     :=  MQTTCLIENTINTERFACE_LOGGING_LEVEL_ERR,
                          dMsgGroup   :=  MQCLIINF_LOG_ERROR_XML_DATAMAP_TE_NAME_LEN_GRP,
                          dMsgNbr     :=  MQCLIINF_LOG_ERROR_XML_DATAMAP_TE_NAME_LEN_MSG,
                          pMsg        :=  MQCLIINF_LOG_ERROR_XML_DATAMAP_TE_NAME_LEN_TEXT,
                          pPara1      :=  #tmpPara,
                          pPara2      :=  NIL,
                          pPara3      :=  NIL,
                          pPara4      :=  NIL);

        return;
      end_if;

      SigCLib.MemSet( dst :=  #aEndpointName,
                    c   :=  0x00,
                    len :=  sizeof(aEndpointName));
      SigCLib.StrCpy( dst0  :=  #aEndpointName[0],
                        src0  :=  pAtt^.Value$^CHAR);
      bNameSet := TRUE;

    //------------------------
    //Element
    //------------------------
    elsif SigCLib.StrCmp(ps1:=#aString[0], ps2:=MQTTCLIENT_INT_XML_DATAMAP_TOPICENDPOINT_ATTR_ELEMENT) = 0 then

      udLen := SigCLib.StrLen(str:=pAtt^.Value$^CHAR);

      if udLen > MQTTCLIENT_INT_XML_DATAMAP_TOPICENDPOINT_ELEMENT_MAX_LEN |
         udLen = 0                                                        then
        //Create Log: DataMap, Element text too long

        Logging_InterfLog(usLevel     :=  MQTTCLIENTINTERFACE_LOGGING_LEVEL_ERR,
                          dMsgGroup   :=  MQCLIINF_LOG_ERROR_XML_DATAMAP_TE_ELEMENT_LEN_GRP,
                          dMsgNbr     :=  MQCLIINF_LOG_ERROR_XML_DATAMAP_TE_ELEMENT_LEN_MSG,
                          pMsg        :=  MQCLIINF_LOG_ERROR_XML_DATAMAP_TE_ELEMENT_LEN_TEXT,
                          pPara1      :=  NIL,
                          pPara2      :=  NIL,
                          pPara3      :=  NIL,
                          pPara4      :=  NIL);

        return;
      end_if;

      SigCLib.MemSet( dst :=  #aElement,
                    c   :=  0x00,
                    len :=  sizeof(aElement));
      SigCLib.StrCpy(dst0:=#aElement[0], src0:=pAtt^.Value$^CHAR);
      bElementSet := TRUE;

    //------------------------
    //Operation
    //------------------------
    elsif SigCLib.StrCmp(ps1:=#aString[0], ps2:=MQTTCLIENT_INT_XML_DATAMAP_TOPICENDPOINT_ATTR_OPERATION) = 0 then

      Operation := ProcessXML_ProcessDataMap_TopicEndpoint_GetOperation(pChar:=pAtt^.Value$^CHAR);
      if Operation = DO_Unknown then
        //Create Log: DataMap, operation type unknown.

        Logging_InterfLog(usLevel     :=  MQTTCLIENTINTERFACE_LOGGING_LEVEL_ERR,
                          dMsgGroup   :=  MQCLIINF_LOG_ERROR_XML_DATAMAP_TE_UNKNOWN_TYPE_GRP,
                          dMsgNbr     :=  MQCLIINF_LOG_ERROR_XML_DATAMAP_TE_UNKNOWN_TYPE_MSG,
                          pMsg        :=  MQCLIINF_LOG_ERROR_XML_DATAMAP_TE_UNKNOWN_TYPE_TEXT,
                          pPara1      :=  NIL,
                          pPara2      :=  NIL,
                          pPara3      :=  NIL,
                          pPara4      :=  NIL);

        return;
      end_if;

    //------------------------
    //Interval
    //------------------------
    elsif SigCLib.StrCmp(ps1:=#aString[0], ps2:=MQTTCLIENT_INT_XML_DATAMAP_TOPICENDPOINT_ATTR_INTERVAL) = 0 then

      udLen := SigCLib.StrLen(str:=pAtt^.Value$^CHAR);

      if udLen > MQTTCLIENT_INT_XML_DATAMAP_TOPICENDPOINT_ATTR_INTERVAL_MAX_LEN then
        //Create Log: DataMap, Interval string too long

        tmpPara := to_dint(udLen);

        Logging_InterfLog(usLevel     :=  MQTTCLIENTINTERFACE_LOGGING_LEVEL_ERR,
                          dMsgGroup   :=  MQCLIINF_LOG_ERROR_XML_DATAMAP_TE_INTERVEL_LEN_GRP,
                          dMsgNbr     :=  MQCLIINF_LOG_ERROR_XML_DATAMAP_TE_INTERVEL_LEN_MSG,
                          pMsg        :=  MQCLIINF_LOG_ERROR_XML_DATAMAP_TE_INTERVEL_LEN_TEXT,
                          pPara1      :=  #tmpPara,
                          pPara2      :=  NIL,
                          pPara3      :=  NIL,
                          pPara4      :=  NIL);

        return;
      end_if;

      udInterval := to_udint(SigCLib.AToI(ps1:=pAtt^.Value$^CHAR));

    //------------------------
    //Datatype
    //------------------------
    elsif SigCLib.StrCmp(ps1:=#aString[0], ps2:=MQTTCLIENT_INT_XML_DATAMAP_TOPICENDPOINT_ATTR_DATATYPE) = 0 then

      DataType := ProcessXML_ProcessDataMap_TopicEndpoint_GetDataType(pChar:=pAtt^.Value$^CHAR);

      if DataType = DD_Unknown then
        //Create Log: DataMap, Datatype unknown.

        Logging_InterfLog(usLevel     :=  MQTTCLIENTINTERFACE_LOGGING_LEVEL_ERR,
                          dMsgGroup   :=  MQCLIINF_LOG_ERROR_XML_DATAMAP_TE_DATATYPE_UNKNOWN_GRP,
                          dMsgNbr     :=  MQCLIINF_LOG_ERROR_XML_DATAMAP_TE_DATATYPE_UNKNOWN_MSG,
                          pMsg        :=  MQCLIINF_LOG_ERROR_XML_DATAMAP_TE_DATATYPE_UNKNOWN_TEXT,
                          pPara1      :=  NIL,
                          pPara2      :=  NIL,
                          pPara3      :=  NIL,
                          pPara4      :=  NIL);

        return;

      end_if;

    //------------------------
    //QoS
    //------------------------
    elsif SigCLib.StrCmp(ps1:=#aString[0], ps2:=MQTTCLIENT_INT_XML_DATAMAP_TOPICENDPOINT_ATTR_QOS) = 0 then

      udLen := SigCLib.StrLen(str:=pAtt^.Value$^CHAR);

      if udLen > MQTTCLIENT_INT_XML_DATAMAP_TOPICENDPOINT_ATTR_QOS_MAX_LEN then
        //Create Log: DataMap, QoS string too long

        tmpPara := to_dint(udLen);

        Logging_InterfLog(usLevel     :=  MQTTCLIENTINTERFACE_LOGGING_LEVEL_ERR,
                          dMsgGroup   :=  MQCLIINF_LOG_ERROR_XML_DATAMAP_TE_QOS_LEN_GRP,
                          dMsgNbr     :=  MQCLIINF_LOG_ERROR_XML_DATAMAP_TE_QOS_LEN_MSG,
                          pMsg        :=  MQCLIINF_LOG_ERROR_XML_DATAMAP_TE_QOS_LEN_TEXT,
                          pPara1      :=  #tmpPara,
                          pPara2      :=  NIL,
                          pPara3      :=  NIL,
                          pPara4      :=  NIL);

        return;
      end_if;

      iQoS := to_int(SigCLib.AToI(ps1:=pAtt^.Value$^CHAR));

      if iQos < MQTT_PROT_QOS_MIN |
         iQoS > MQTT_PROT_QOS_MAX then
        //Create Log: DataMap, QoS Invalid

        tmpPara := to_dint(iQoS);

        Logging_InterfLog(usLevel     :=  MQTTCLIENTINTERFACE_LOGGING_LEVEL_ERR,
                          dMsgGroup   :=  MQCLIINF_LOG_ERROR_XML_DATAMAP_TE_QOS_INVALID_GRP,
                          dMsgNbr     :=  MQCLIINF_LOG_ERROR_XML_DATAMAP_TE_QOS_INVALID_MSG,
                          pMsg        :=  MQCLIINF_LOG_ERROR_XML_DATAMAP_TE_QOS_INVALID_TEXT,
                          pPara1      :=  #tmpPara,
                          pPara2      :=  NIL,
                          pPara3      :=  NIL,
                          pPara4      :=  NIL);

        return;
      end_if;

    //------------------------
    //Retain
    //------------------------
    elsif SigCLib.StrCmp(ps1:=#aString[0], ps2:=MQTTCLIENT_INT_XML_DATAMAP_TOPICENDPOINT_ATTR_RETAIN) = 0 then

      udLen := SigCLib.StrLen(str:=pAtt^.Value$^CHAR);

      if udLen > MQTTCLIENT_INT_XML_DATAMAP_TOPICENDPOINT_ATTR_RETAIN_MAX_LEN then
        //Create Log: DataMap, Retin String too long

        Logging_InterfLog(usLevel     :=  MQTTCLIENTINTERFACE_LOGGING_LEVEL_ERR,
                          dMsgGroup   :=  MQCLIINF_LOG_ERROR_XML_DATAMAP_TE_RETAIN_LEN_GRP,
                          dMsgNbr     :=  MQCLIINF_LOG_ERROR_XML_DATAMAP_TE_RETAIN_LEN_MSG,
                          pMsg        :=  MQCLIINF_LOG_ERROR_XML_DATAMAP_TE_RETAIN_LEN_TEXT,
                          pPara1      :=  NIL,
                          pPara2      :=  NIL,
                          pPara3      :=  NIL,
                          pPara4      :=  NIL);

      end_if;

      DRSRetain := ProcessXML_ProcessDataMap_TopicEndpoint_GetRetain(pChar:=pAtt^.Value$^CHAR);

      if DRSRetain = DRS_Unknown then
        //Create Log: DataMap, Retain Value not known.

        Logging_InterfLog(usLevel     :=  MQTTCLIENTINTERFACE_LOGGING_LEVEL_ERR,
                          dMsgGroup   :=  MQCLIINF_LOG_ERROR_XML_DATAMAP_TE_RETAIN_INVALID_GRP,
                          dMsgNbr     :=  MQCLIINF_LOG_ERROR_XML_DATAMAP_TE_RETAIN_INVALID_MSG,
                          pMsg        :=  MQCLIINF_LOG_ERROR_XML_DATAMAP_TE_RETAIN_INVALID_TEXT,
                          pPara1      :=  #DRSRetain$DINT,
                          pPara2      :=  NIL,
                          pPara3      :=  NIL,
                          pPara4      :=  NIL);

        return;

      end_if;

    end_if;

    udAtt -= 1;

  end_while;

  //OK If the Name and element are set
  bOK := bNameSet & bElementSet;

  //Required Elements set
  if bOK then

    SigCLib.MemSet( dst :=  #aTopicString[0],
                    c   :=  0x00,
                    len :=  sizeof(aTopicString));

    udCount := 0;

    //Build the Topic String (Concatenate all the Sections and Endpoint).
    while udCount < Config.pDataMapConfig^.udTopicStringDepth do

      udLen := SigCLib.StrLen(str:=#Config.pDataMapConfig^.aTopicStrings[udCount][0]) + SigCLib.StrLen(str:=#aTopicString[0]) + 1;

      //String will fit
      if udLen < MQTTCLIENT_TOPIC_MAX_LEN then

        if udCount > 0 then

          SigCLib.StrCat( ps1  :=  #aTopicString[0],
                          ps2  :=  MQTTCLIENT_INT_XML_DATAMAP_TOPIC_DIVIDER);
        end_if;

        SigCLib.StrCat( ps1  :=  #aTopicString[0],
                        ps2  :=  #Config.pDataMapConfig^.aTopicStrings[udCount][0]);

      //String too long
      else

        tmpPara := to_dint(udLen);

        //Create Log: Topic too long
        Logging_InterfLog(usLevel     :=  MQTTCLIENTINTERFACE_LOGGING_LEVEL_ERR,
                          dMsgGroup   :=  MQCLIINF_LOG_ERROR_XML_DATAMAP_TE_TOPIC_LEN_GRP,
                          dMsgNbr     :=  MQCLIINF_LOG_ERROR_XML_DATAMAP_TE_TOPIC_LEN_MSG,
                          pMsg        :=  MQCLIINF_LOG_ERROR_XML_DATAMAP_TE_TOPIC_LEN_TEXT,
                          pPara1      :=  NIL,
                          pPara2      :=  NIL,
                          pPara3      :=  NIL,
                          pPara4      :=  NIL);

        return;

      end_if;

      udCount += 1;

    end_while;

    if Config.pDataMapConfig^.udTopicStringDepth > 0                          &
       SigCLib.StrLen(str:=#aTopicString[0]) + 1 <= MQTTCLIENT_TOPIC_MAX_LEN  then

      SigCLib.StrCat( ps1  :=  #aTopicString[0],
                      ps2  :=  MQTTCLIENT_INT_XML_DATAMAP_TOPIC_DIVIDER);

    end_if;

    udLen := SigCLib.StrLen(str:=#aTopicString[0]) + SigCLib.StrLen(str:=#aEndpointName[0]);

    if udLen >= MQTTCLIENT_TOPIC_MAX_LEN then
      //Create Log: DataMap Processing Element Failed, topic name too long

      tmpPara := to_dint(udLen);

      Logging_InterfLog(usLevel     :=  MQTTCLIENTINTERFACE_LOGGING_LEVEL_ERR,
                        dMsgGroup   :=  MQCLIINF_LOG_ERROR_XML_DATAMAP_TE_CONCAT_TOPIC_LEN_GRP,
                        dMsgNbr     :=  MQCLIINF_LOG_ERROR_XML_DATAMAP_TE_CONCAT_TOPIC_LEN_MSG,
                        pMsg        :=  MQCLIINF_LOG_ERROR_XML_DATAMAP_TE_CONCAT_TOPIC_LEN_TEXT,
                        pPara1      :=  #tmpPara,
                        pPara2      :=  NIL,
                        pPara3      :=  NIL,
                        pPara4      :=  NIL);

      bOK := FALSE;
      return;
    end_if;

    SigCLib.StrCat( ps1 :=  #aTopicString[0],
                    ps2 :=  #aEndpointName[0]);

    DataMapRet := DataMap_AddElement_Internal(pTopic      :=  #aTopicString[0],
                                              pElement    :=  #aElement[0],
                                              Operation   :=  Operation,
                                              Datatype    :=  DataType,
                                              udInterval  :=  udInterval,
                                              iQoS        :=  iQos,
                                              bRetain     :=  (DRSRetain = DRS_True),
                                              bAddedByXML :=  TRUE);

    bOK := DataMapRet = DM_OK;

    if bOK = FALSE then

      //Create Log: DataMap, adding Element to DataMap Failed.
      Logging_InterfLog(usLevel     :=  MQTTCLIENTINTERFACE_LOGGING_LEVEL_ERR,
                        dMsgGroup   :=  MQCLIINF_LOG_ERROR_XML_DATAMAP_TE_DATAMAP_ADD_FAIL_GRP,
                        dMsgNbr     :=  MQCLIINF_LOG_ERROR_XML_DATAMAP_TE_DATAMAP_ADD_FAIL_MSG,
                        pMsg        :=  MQCLIINF_LOG_ERROR_XML_DATAMAP_TE_DATAMAP_ADD_FAIL_TEXT,
                        pPara1      :=  #DataMapRet$DINT,
                        pPara2      :=  NIL,
                        pPara3      :=  NIL,
                        pPara4      :=  NIL);

      return;
    end_if;

  //Required Elements not set
  else

    //Create Log: DataMap, Failed processing topic endpoint, all required attributes have not been set

    Logging_InterfLog(usLevel     :=  MQTTCLIENTINTERFACE_LOGGING_LEVEL_ERR,
                      dMsgGroup   :=  MQCLIINF_LOG_ERROR_XML_DATAMAP_TE_MISSING_ENTRIES_GRP,
                      dMsgNbr     :=  MQCLIINF_LOG_ERROR_XML_DATAMAP_TE_MISSING_ENTRIES_MSG,
                      pMsg        :=  MQCLIINF_LOG_ERROR_XML_DATAMAP_TE_MISSING_ENTRIES_TEXT,
                      pPara1      :=  NIL,
                      pPara2      :=  NIL,
                      pPara3      :=  NIL,
                      pPara4      :=  NIL);

    return;

  end_if;

END_FUNCTION

FUNCTION MQTTClient_Interface::ProcessXML_ProcessDataMap_TopicEndpoint_GetOperation
	VAR_INPUT
		pChar 	: ^CHAR;
	END_VAR
	VAR_OUTPUT
		Operation 	: t_e_DataMap_Operations;
	END_VAR
  VAR
  	aString : ARRAY[0..MQTTCLIENT_INT_XML_DATAMAP_TOPICENDPOINT_OPERATION_MAX_LEN] of CHAR;
  END_VAR

  //Assume not found
  Operation := DO_Unknown;

  if pChar = NIL then
    return;
  end_if;

  //Convert the String to all upper for comparison to eliminate casing constraints
    SigCLib.StrNCpy(dst0  :=  #aString[0],
                    src0  :=  pChar,
                    count :=  MQTTCLIENT_INT_XML_DATAMAP_TOPICENDPOINT_OPERATION_MAX_LEN-1);

    aString[SigCLib.StrLen(str:=pChar)] := 0x00;

    SigCLib.StrUpr(ps1:=#aString[0]);

  //Poll
  if SigCLib.StrCmp(ps1:=#aString[0], ps2:=MQTTCLIENT_INT_XML_DATAMAP_TOPICENDPOINT_OPERATION_POLL) = 0 then

    Operation := DO_Poll;

  //Change
  elsif SigCLib.StrCmp(ps1:=#aString[0], ps2:=MQTTCLIENT_INT_XML_DATAMAP_TOPICENDPOINT_OPERATION_CHANGE) = 0 then

    Operation := DO_Change;

  //Subscribe
  elsif SigCLib.StrCmp(ps1:=#aString[0], ps2:=MQTTCLIENT_INT_XML_DATAMAP_TOPICENDPOINT_OPERATION_SUBSCRIBE) = 0 then

    Operation := DO_Subscribe;

  end_if;

END_FUNCTION

FUNCTION MQTTClient_Interface::ProcessXML_ProcessDataMap_TopicEndpoint_GetDataType
	VAR_INPUT
		pChar 	: ^CHAR;
	END_VAR
	VAR_OUTPUT
		DataType 	: t_e_DataMap_DataTypes;
	END_VAR
  VAR
  	aString : ARRAY[0..MQTTCLIENT_INT_XML_DATAMAP_TOPICENDPOINT_DATATYPE_MAXLEN] of CHAR;
  END_VAR

  //Assume not found
  DataType := DD_Unknown;

  if pChar = NIL then
    return;
  end_if;

  //Convert the String to all upper for comparison to eliminate casing constraints
    SigCLib.StrNCpy(dst0  :=  #aString[0],
                    src0  :=  pChar,
                    count :=  MQTTCLIENT_INT_XML_DATAMAP_TOPICENDPOINT_DATATYPE_MAXLEN-1);

    aString[SigCLib.StrLen(str:=pChar)] := 0x00;

    SigCLib.StrUpr(ps1:=#aString[0]);

  //DINT
  if SigCLib.StrCmp(ps1:=#aString[0], ps2:=MQTTCLIENT_INT_XML_DATAMAP_TOPICENDPOINT_DATATYPE_DINT) = 0 then

    DataType := DD_DINT;

  //UDINT
  elsif SigCLib.StrCmp(ps1:=#aString[0], ps2:=MQTTCLIENT_INT_XML_DATAMAP_TOPICENDPOINT_DATATYPE_UDINT) = 0 then

    DataType := DD_UDINT;

  //REAL
  elsif SigCLib.StrCmp(ps1:=#aString[0], ps2:=MQTTCLIENT_INT_XML_DATAMAP_TOPICENDPOINT_DATATYPE_REAL) = 0 then

    DataType := DD_REAL;

  //String
  elsif SigCLib.StrCmp(ps1:=#aString[0], ps2:=MQTTCLIENT_INT_XML_DATAMAP_TOPICENDPOINT_DATATYPE_STRING) = 0 then

    DataType := DD_STRING;

  end_if;

END_FUNCTION

FUNCTION MQTTClient_Interface::ProcessXML_ProcessDataMap_TopicEndpoint_GetRetain
	VAR_INPUT
		pChar 	: ^CHAR;
	END_VAR
	VAR_OUTPUT
		RetainState 	: t_e_DataMap_RetainStates;
	END_VAR
  VAR
  	aString : ARRAY[0..MQTTCLIENT_INT_XML_DATAMAP_TOPICENDPOINT_RETAIN_MAX_LEN] of CHAR;
  END_VAR

  //Assume not found
  RetainState := DRS_Unknown;

  if pChar = NIL then
    return;
  end_if;

  //Convert the String to all upper for comparison to eliminate casing constraints
    SigCLib.StrNCpy(dst0  :=  #aString[0],
                    src0  :=  pChar,
                    count :=  MQTTCLIENT_INT_XML_DATAMAP_TOPICENDPOINT_RETAIN_MAX_LEN-1);

    aString[SigCLib.StrLen(str:=pChar)] := 0x00;

    SigCLib.StrUpr(ps1:=#aString[0]);

  //TRUE
  if SigCLib.StrCmp(ps1:=#aString[0], ps2:=MQTTCLIENT_INT_XML_DATAMAP_TOPICENDPOINT_RETAIN_TRUE) = 0 then

    RetainState := DRS_True;

  //FALSE
  elsif SigCLib.StrCmp(ps1:=#aString[0], ps2:=MQTTCLIENT_INT_XML_DATAMAP_TOPICENDPOINT_RETAIN_FALSE) = 0 then

    RetainState := DRS_False;

  end_if;

END_FUNCTION
//================================================================================================================================================================
//------------------------------------------------------------------END OF PROCESS XML METHODS--------------------------------------------------------------------
//================================================================================================================================================================

//================================================================================================================================================================
//----------------------------------------------------------------------DATAMAP METHODS---------------------------------------------------------------------------
//================================================================================================================================================================
FUNCTION MQTTClient_Interface::DataMap_AddElement
	VAR_INPUT
		pTopic 	: ^CHAR;
		pElement 	: ^CHAR;
		Operation 	: t_e_DataMap_Operations;
		Datatype 	: t_e_DataMap_DataTypes;
		udInterval 	: UDINT;
		iQoS 	: INT;
		bRetain 	: BOOL;
	END_VAR
	VAR_OUTPUT
		RetCode 	: t_e_DataMap_RetCode;
	END_VAR

  RetCode := DataMap_AddElement_Internal(pTopic, pElement, Operation, Datatype, udInterval, iQoS, bRetain, bAddedByXML:=FALSE);

END_FUNCTION

FUNCTION MQTTClient_Interface::DataMap_AddElement_Internal
	VAR_INPUT
		pTopic 	: ^CHAR;
		pElement 	: ^CHAR;
		Operation 	: t_e_DataMap_Operations;
		Datatype 	: t_e_DataMap_DataTypes;
		udInterval 	: UDINT;
		iQoS 	: INT;
		bRetain 	: BOOL;
		bAddedByXML 	: BOOL;
	END_VAR
	VAR_OUTPUT
		RetCode 	: t_e_DataMap_RetCode;
	END_VAR
  VAR
  	pElementPtr : ^void;
    ChannelMode : CHMODE;
    pPubEntry   : ^t_s_DataMap_ElementEntry_Publish;
    pSubEntry   : ^t_s_DataMap_ElementEntry_Subscribe;
    tmpPara1    : DINT;
    udLen       : UDINT;
  END_VAR

  RetCode := DM_OK;

  if pTopic = NIL           |
     pElement = NIL         |
     Datatype = DD_Unknown  |
     Operation = DO_Unknown then

    RetCode := DM_InputValueError;
    //Create Log: Adding DataMap Element failed, Inout value error

    Logging_InterfLog(usLevel     :=  MQTTCLIENTINTERFACE_LOGGING_LEVEL_ERR,
                      dMsgGroup   :=  MQCLIINF_LOG_ERROR_DATAMAP_ADD_FAIL_INPUT_GRP,
                      dMsgNbr     :=  MQCLIINF_LOG_ERROR_DATAMAP_ADD_FAIL_INPUT_MSG,
                      pMsg        :=  MQCLIINF_LOG_ERROR_DATAMAP_ADD_FAIL_INPUT_TEXT,
                      pPara1      :=  NIL,
                      pPara2      :=  NIL,
                      pPara3      :=  NIL,
                      pPara4      :=  NIL);

    return;

  end_if;

  //Check Topic Name Len
  udLen := SigCLib.StrLen(str:=pTopic);

  if udLen >= MQTTCLIENTINTERFACE_DATAMAP_TOPIC_NAME_MAX_LEN then

    RetCode := DM_TopicNameTooLong;
    //Create Log: Adding Publish Element Failed, Topic Name too long

    tmpPara1 := to_dint(udLen);

    Logging_InterfLog(usLevel     :=  MQTTCLIENTINTERFACE_LOGGING_LEVEL_ERR,
                      dMsgGroup   :=  MQCLIINF_LOG_ERROR_DATAMAP_ADD_FAIL_TOPIC_LEN_GRP,
                      dMsgNbr     :=  MQCLIINF_LOG_ERROR_DATAMAP_ADD_FAIL_TOPIC_LEN_MSG,
                      pMsg        :=  MQCLIINF_LOG_ERROR_DATAMAP_ADD_FAIL_TOPIC_LEN_TEXT,
                      pPara1      :=  #tmpPara1,
                      pPara2      :=  NIL,
                      pPara3      :=  NIL,
                      pPara4      :=  NIL);

    return;

  end_if;

  udLen := SigCLib.StrLen(str:=pElement);

  if udLen >= MQTTCLIENTINTERFACE_DATAMAP_ELEMENT_MAX_LEN then

    RetCode := DM_ElementNameTooLong;
    //Create Log: Adding Publish Element Failed, Element Name too long

    tmpPara1 := to_dint(udLen);

    Logging_InterfLog(usLevel     :=  MQTTCLIENTINTERFACE_LOGGING_LEVEL_ERR,
                      dMsgGroup   :=  MQCLIINF_LOG_ERROR_DATAMAP_ADD_FAIL_ELEMENT_LEN_GRP,
                      dMsgNbr     :=  MQCLIINF_LOG_ERROR_DATAMAP_ADD_FAIL_ELEMENT_LEN_MSG,
                      pMsg        :=  MQCLIINF_LOG_ERROR_DATAMAP_ADD_FAIL_ELEMENT_LEN_TEXT,
                      pPara1      :=  #tmpPara1,
                      pPara2      :=  NIL,
                      pPara3      :=  NIL,
                      pPara4      :=  NIL);

    return;

  end_if;

  ChannelMode := _LookUpEmbed_C(  pText   :=  pElement,
                                  pObj_ch :=  #pElementPtr,
                                  pObj    :=  NIL);

  //If the Pointer is not found, log and fail
  if pElementPtr = NIL then

    RetCode := DM_ElementNotFound;
    //Create Log: Adding DataMap Element failed, Element not found

    Logging_InterfLog(usLevel     :=  MQTTCLIENTINTERFACE_LOGGING_LEVEL_ERR,
                      dMsgGroup   :=  MQCLIINF_LOG_ERROR_DATAMAP_ADD_FAIL_NOT_FOUND_GRP,
                      dMsgNbr     :=  MQCLIINF_LOG_ERROR_DATAMAP_ADD_FAIL_NOT_FOUND_MSG,
                      pMsg        :=  MQCLIINF_LOG_ERROR_DATAMAP_ADD_FAIL_NOT_FOUND_TEXT,
                      pPara1      :=  NIL,
                      pPara2      :=  NIL,
                      pPara3      :=  NIL,
                      pPara4      :=  NIL);

    return;

  //If the Channel type is not OK, log & Fail
    //If this is a String and the ChannelType is not Object
    //If this is a 4-Byte Value and the ChannelTye is not SVR and not CMD.
  elsif (Datatype = DD_String   &
        ChannelMode <> _CH_OBJ) |
        ((Datatype = DD_DINT   |
          Datatype = DD_UDINT  |
          Datatype = DD_REAL)  &
         (ChannelMode <> _CH_SVR) &
         (ChannelMode <> _CH_CMD)) then

    RetCode := DM_InputValueError;

    //Create Log:
    Logging_InterfLog(usLevel     :=  MQTTCLIENTINTERFACE_LOGGING_LEVEL_ERR,
                      dMsgGroup   :=  MQCLIINF_LOG_ERROR_DATAMAP_ADD_FAIL_TYPE_MISMATCH_GRP,
                      dMsgNbr     :=  MQCLIINF_LOG_ERROR_DATAMAP_ADD_FAIL_TYPE_MISMATCH_MSG,
                      pMsg        :=  MQCLIINF_LOG_ERROR_DATAMAP_ADD_FAIL_TYPE_MISMATCH_TEXT,
                      pPara1      :=  NIL,
                      pPara2      :=  NIL,
                      pPara3      :=  NIL,
                      pPara4      :=  NIL);

    return;

  end_if;

  //==============================================================
  //Based on the requested operation, add the element to the list
  //==============================================================
  case Operation of
    //---------------------------------
    //PUBLISH
  	//---------------------------------
    t_e_DataMap_Operations::DO_Poll, DO_Change:

      if Config.pDataMapConfig^.udPublishElements >= Config.pDataMapConfig^.udEntries then

        RetCode := DM_ListFull;
        //Create Log: Adding Publish Element Failed, Too many entries

        Logging_InterfLog(usLevel     :=  MQTTCLIENTINTERFACE_LOGGING_LEVEL_ERR,
                          dMsgGroup   :=  MQCLIINF_LOG_ERROR_DATAMAP_ADD_PUB_FAIL_FULL_GRP,
                          dMsgNbr     :=  MQCLIINF_LOG_ERROR_DATAMAP_ADD_PUB_FAIL_FULL_MSG,
                          pMsg        :=  MQCLIINF_LOG_ERROR_DATAMAP_ADD_PUB_FAIL_FULL_TEXT,
                          pPara1      :=  NIL,
                          pPara2      :=  NIL,
                          pPara3      :=  NIL,
                          pPara4      :=  NIL);

        return;

      end_if;

      pPubEntry := (Config.pDataMapConfig^.Elements.pPublishEntries$UDINT + (sizeof(t_s_DataMap_ElementEntry_Publish)*Config.pDataMapConfig^.udPublishElements))$^t_s_DataMap_ElementEntry_Publish;
      //pPubEntry := #Config.pDataMapConfig^.Elements.aPublishEntries[Config.pDataMapConfig^.udPublishElements];

      pPubEntry^.pData         := pElementPtr;
      pPubEntry^.Operation     := Operation;
      pPubEntry^.Datatype      := Datatype;
      pPubEntry^.iQoS          := iQoS;
      pPubEntry^.bRetain       := bRetain;
      pPubEntry^.udInterval    := udInterval;
      pPubEntry^.udLastAction  := ops.tAbsolute;
      pPubEntry^.bAddedByXML   := bAddedByXML;
      pPubEntry^.pTempMem      := NIL;

      SigCLib.MemSet( dst :=  #pPubEntry^.aElement,
                      c   :=  0x00,
                      len :=  MQTTCLIENT_INT_XML_DATAMAP_TOPICENDPOINT_ELEMENT_MAX_LEN);

      SigCLib.StrCpy( dst0  :=  #pPubEntry^.aElement[0],
                      src0  :=  pElement);

      SigCLib.MemSet( dst   :=  #pPubEntry^.aTopic,
                      c     :=  0x00,
                      len   :=  sizeof(t_s_DataMap_ElementEntry_Publish.aTopic));

      SigCLib.Utf8ToStr16(dst := #pPubEntry^.aTopic[0],
                          src := pTopic);

      pPubEntry^.udDataLen  := 0;
      pPubEntry^.udCRC      := 0;
      //===================================
      //Based on Type, set Len
      //===================================
      case Datatype of
      	t_e_DataMap_DataTypes::DD_UDINT:
          pPubEntry^.udDataLen := MQTTCLIENTINTERFACE_DATAMAP_DATALEN_UDINT;
      	t_e_DataMap_DataTypes::DD_DINT:
          pPubEntry^.udDataLen := MQTTCLIENTINTERFACE_DATAMAP_DATALEN_DINT;
      	t_e_DataMap_DataTypes::DD_REAL:
          pPubEntry^.udDataLen := MQTTCLIENTINTERFACE_DATAMAP_DATALEN_REAL;
      end_case;

      //Calc CRC
      if Operation = DO_Change then

        // If the value should not be published immediately, we set the flag to true so that the initial publish is not made
        pPubEntry^.bInitialPublish := Config.pDataMapConfig^.Config.bSendOnAdd = FALSE;

        if  pPubEntry^.udDataLen > 0           &
            pPubEntry^.Datatype <> DD_String  then

          pPubEntry^.udCRC$DINT := RD(pt:= pPubEntry^.pData);

        elsif pPubEntry^.Datatype = DD_String then

          pPubEntry^.udCRC := pPubEntry^.pData$^StringInternal^.GetCRC();

        end_if;

      end_if;

      pPubEntry^.State := DMPS_Ready;
      Config.pDataMapConfig^.udPublishElements += 1;

    //---------------------------------
    //Subscribe
    //---------------------------------
  	t_e_DataMap_Operations::DO_Subscribe:

      if Config.pDataMapConfig^.udSubscribeElements >= Config.pDataMapConfig^.udEntries then
        RetCode := DM_ListFull;
        //Create Log: Adding Subscribe Element Failed, Too many entries

        tmpPara1 := to_dint(Config.pDataMapConfig^.udEntries);

        Logging_InterfLog(usLevel     :=  MQTTCLIENTINTERFACE_LOGGING_LEVEL_ERR,
                          dMsgGroup   :=  MQCLIINF_LOG_ERROR_DATAMAP_ADD_SUB_FAIL_FULL_GRP,
                          dMsgNbr     :=  MQCLIINF_LOG_ERROR_DATAMAP_ADD_SUB_FAIL_FULL_MSG,
                          pMsg        :=  MQCLIINF_LOG_ERROR_DATAMAP_ADD_SUB_FAIL_FULL_TEXT,
                          pPara1      :=  NIL,
                          pPara2      :=  NIL,
                          pPara3      :=  NIL,
                          pPara4      :=  NIL);

        return;
      end_if;

      pSubEntry := (Config.pDataMapConfig^.Elements.pSubscribeEntries$UDINT + (sizeof(t_s_DataMap_ElementEntry_Subscribe)*Config.pDataMapConfig^.udSubscribeElements))$^t_s_DataMap_ElementEntry_Subscribe;
      //pSubEntry := #Config.pDataMapConfig^.Elements.aSubscribeEntries[Config.pDataMapConfig^.udSubscribeElements];

      pSubEntry^.pData        := pElementPtr;
      pSubEntry^.Datatype     := Datatype;
      pSubEntry^.iQoS         := iQoS;
      pSubEntry^.bAddedByXML  := bAddedByXML;
      pSubEntry^.bRemove      := FALSE;

      SigCLib.MemSet( dst :=  #pSubEntry^.aElement,
                      c   :=  0x00,
                      len :=  MQTTCLIENT_INT_XML_DATAMAP_TOPICENDPOINT_ELEMENT_MAX_LEN);

      SigCLib.StrCpy( dst0  :=  #pSubEntry^.aElement[0],
                      src0  :=  pElement);

      SigCLib.MemSet( dst   :=  #pSubEntry^.aTopic,
                      c     :=  0x00,
                      len   :=  sizeof(t_s_DataMap_ElementEntry_Subscribe.aTopic));

      SigCLib.Utf8ToStr16(dst := #pSubEntry^.aTopic[0],
                          src := pTopic);

      pSubEntry^.State := DMSS_Ready;
      Config.pDataMapConfig^.udSubscribeElements += 1;

  end_case;

  RetCode := DM_OK;

END_FUNCTION

FUNCTION MQTTClient_Interface::DataMap_ProcessMap

  //Process the DataMap Lists
  DataMap_ProcessMap_Publish();
  DataMap_ProcessMap_Subscribe();

END_FUNCTION

FUNCTION MQTTClient_Interface::DataMap_ProcessMap_Publish
  VAR
  	pEntry    : ^t_s_DataMap_ElementEntry_Publish;
    udCount   : UDINT;
    pData     : ^void;
    tmpPara1  : DINT;
    tmpPara2  : DINT;
    iMQRet    : INT;
  END_VAR

  //Process the Publish List
  if Config.pDataMapConfig^.udPublishElements > 0 then

    for udCount := 0 to Config.pDataMapConfig^.udPublishElements - 1 do

      pEntry := (Config.pDataMapConfig^.Elements.pPublishEntries$UDINT + (udCount*sizeof(t_s_DataMap_ElementEntry_Publish)))$^t_s_DataMap_ElementEntry_Publish;

      //=========================================================
      //Entry FSM
      //=========================================================
      case pEntry^.State of
        //--------------------------------------------
        //Prepare
        //--------------------------------------------
        t_e_DataMap_PublishStates::DMPS_Ready:

          pEntry^.udLastAction := ops.tAbsolute;
          pEntry^.State := DMPS_WaitForAction;

        //--------------------------------------------
        //Wait for publish event
        //--------------------------------------------
        t_e_DataMap_PublishStates::DMPS_WaitForAction:

          //If the entry needs to be removed, remove it
          if pEntry^.bRemove then

            pEntry^.State := DMPS_Remove;
            return;

          end_if;

          //Reset MID
          pEntry^.iMid := -1;

          //Test for Timeout (or if the initial publish should be made)
          if ops.tAbsolute - pEntry^.udLastAction >= pEntry^.udInterval
            | pEntry^.bInitialPublish = FALSE then

            //Test for Event and prepare to send

            //Poll always sends, advance to publish
            if pEntry^.Operation = DO_Poll then

              pEntry^.State := DMPS_Publish;

            //If the data needs to be monitored for a change, check if changed and advance to publish if necessary
            elsif pEntry^.Operation = DO_Change then

              //Determine if the data has changed

                //If this is a String object, use the string object CRC method
                if pEntry^.Datatype = DD_String then

                  Config.pDataMapConfig^.udCRC := pEntry^.pData$^StringInternal^.GetCRC();

                //If this is a Server Value, call the Read Method, check if changed and store the value to publish
                elsif pEntry^.Datatype = DD_DINT  |
                      pEntry^.Datatype = DD_UDINT |
                      pEntry^.Datatype = DD_REAL  then

                  //As the CRC and the data is the same length, just read the actual data, we won't unnecessarily calculate a CRC.
                  Config.pDataMapConfig^.udCRC$DINT := RD(pt:= pEntry^.pData);

                //If this is some other block of Data, calculate the CRC Manually
                else

                  Config.pDataMapConfig^.udCRC := sigclib_crc32(  initval :=  MQTTCLIENTINTERFACE_DATAMAP_CRCCALC_INITVAL,
                                                                  psrc    :=  pEntry^.pData,
                                                                  length  :=  pEntry^.udDataLen);
                end_if;

                //Compare the CRCs (Old vs New)
                if pEntry^.udCRC <> Config.pDataMapConfig^.udCRC |
                   pEntry^.bInitialPublish = FALSE               then

                  pEntry^.udCRC := Config.pDataMapConfig^.udCRC;
                  pEntry^.State := DMPS_Publish;

                end_if;

            end_if;

            //Prepare the data to send: If the state was advanced to publish (In the above If-Stetment) We need to collect the data for the publish step
            if pEntry^.State = DMPS_Publish then

              //======================================================================================
              //Based on the DataType, prepare for publishing
              //======================================================================================
              case pEntry^.Datatype of

                //---------------------
                //String Object
                //---------------------
                DD_String:

                  pEntry^.udDataLen := pEntry^.pData$^StringInternal^.GetLength();

                  if pEntry^.udDataLen > MQTTCLIENT_MAX_DATA_LEN then
                    //Create Log: DataMap tried sending a string that is larger than allowable maximum.

                    tmpPara1 := to_dint(pEntry^.udDataLen);
                    tmpPara2 := MQTTCLIENT_MAX_DATA_LEN;

                    Logging_InterfLog(usLevel     :=  MQTTCLIENTINTERFACE_LOGGING_LEVEL_WARNING,
                                      dMsgGroup   :=  MQCLIINF_LOG_WARNING_DATAMAP_STRING_TRUNCATED_GRP,
                                      dMsgNbr     :=  MQCLIINF_LOG_WARNING_DATAMAP_STRING_TRUNCATED_MSG,
                                      pMsg        :=  MQCLIINF_LOG_WARNING_DATAMAP_STRING_TRUNCATED_TEXT,
                                      pPara1      :=  #tmpPara2,
                                      pPara2      :=  #tmpPara1,
                                      pPara3      :=  NIL,
                                      pPara4      :=  NIL);

                    pEntry^.udDataLen := MQTTCLIENT_MAX_DATA_LEN;

                  end_if;

                  if pEntry^.pTempMem <> NIL then

                    //Create Log: DataMap entry Temp Memory POinter was not NIL, Attempting free.
                    tmpPara1 := to_dint(pEntry^.iMid);

                    Logging_InterfLog(usLevel     :=  MQTTCLIENTINTERFACE_LOGGING_LEVEL_WARNING,
                                      dMsgGroup   :=  MQCLIINF_LOG_WARNING_DATAMAP_PUBLISH_TMPPTR_NOTNIL_GRP,
                                      dMsgNbr     :=  MQCLIINF_LOG_WARNING_DATAMAP_PUBLISH_TMPPTR_NOTNIL_MSG,
                                      pMsg        :=  MQCLIINF_LOG_WARNING_DATAMAP_PUBLISH_TMPPTR_NOTNIL_TEXT,
                                      pPara1      :=  #tmpPara1,
                                      pPara2      :=  NIL,
                                      pPara3      :=  NIL,
                                      pPara4      :=  NIL);

                    MQTTClient.Free(mptr:=pEntry^.pTempMem);
                    pEntry^.pTempMem := NIL;

                  end_if;

                  if pEntry^.udDataLen > 0 then

                    // There is some data available, this needs to be copied

                    pEntry^.pTempMem := MQTTClient.MallocV1(size0 :=  pEntry^.udDataLen,
                                                            mark0 :=  MQTTCLIENT_DEFAULT_MALLOC_MARK);

                    if pEntry^.pTempMem = NIL then
                      //Create Log: DataMap failed to allocate memory to send the string: ...

                      tmpPara1 := to_dint(pEntry^.iMid);
                      tmpPara2 := pEntry^.pData$DINT;

                      Logging_InterfLog(usLevel     :=  MQTTCLIENTINTERFACE_LOGGING_LEVEL_ERR,
                                        dMsgGroup   :=  MQCLIINF_LOG_ERROR_DATAMAP_PUBLISH_FAIL_STRMALLOC_GRP,
                                        dMsgNbr     :=  MQCLIINF_LOG_ERROR_DATAMAP_PUBLISH_FAIL_STRMALLOC_MSG,
                                        pMsg        :=  MQCLIINF_LOG_ERROR_DATAMAP_PUBLISH_FAIL_STRMALLOC_TEXT,
                                        pPara1      :=  #tmpPara1,
                                        pPara2      :=  #tmpPara2,
                                        pPara3      :=  NIL,
                                        pPara4      :=  NIL);

                      pEntry^.State := DMPS_WaitForAction;

                    else

                      //We do not care about the 0-Termination of the string as the MQTTClient::Publish() Method will only copy the length specified.
                      pEntry^.pData$^StringInternal^.ReadDataOff( udOff :=  0,
                                                                  pData :=  pEntry^.pTempMem$^USINT,
                                                                  udMax :=  pEntry^.udDataLen);
                    end_if;

                  end_if;

                //---------------------
                //4 Byte Server Values
                //---------------------
                DD_DINT,
                DD_UDINT,
                DD_REAL:

                  //If the server is polled, we still need to fetch the data, do so.
                  if pEntry^.Operation = DO_Poll then

                    pEntry^.TempMem$DINT := RD(pt:=pEntry^.pData);

                  //This is an OnChange-Entry - Server has already been read, do not call the RD() method twice.
                  else

                    //Copy the CRC Value
                    pEntry^.TempMem := pEntry^.udCRC;

                  end_if;

                //--------------------------------------------------------------------------------------------------------------------
                //Other Payloads (Assumed to be a problem, DataMap could be expanded later to fetch blocks of memory behind pointers).
                //--------------------------------------------------------------------------------------------------------------------
                DD_Unknown:

                  pEntry^.State := DMPS_Error;

              end_case;

            end_if;

            //Update the timestamp to be able to wait another cycle
            pEntry^.udLastAction := ops.tAbsolute;

          end_if;

        //--------------------------------------------
        //Perform Publish
        //--------------------------------------------
        t_e_DataMap_PublishStates::DMPS_Publish:

          //Prepare Data pointer
            //Strings are copied into Temporary Memory
            if pEntry^.Datatype = DD_String then

              pData := pEntry^.pTempMem;

            //4-Byte Values are stored in the Structure
            elsif pEntry^.Datatype = DD_DINT  |
                  pEntry^.Datatype = DD_UDINT |
                  pEntry^.Datatype = DD_REAL  then

              pData := #pEntry^.TempMem;

            end_if;

          //Perform Publish
          iMQRet := MQTT_Publish( pTopic        :=  #pEntry^.aTopic[0],
                                  iQoS          :=  pEntry^.iQoS,
                                  pPayload      :=  pData,
                                  udPayloadLen  :=  pEntry^.udDataLen,
                                  bRetain       :=  pEntry^.bRetain,
                                  pThis         :=  this,
                                  pCallback     :=  #DataMap_Return_Callback(),
                                  pMid          :=  #pEntry^.iMid,
                                  pApplMsgID    :=  #pEntry^.udApplID);

          if iMQRet = MQTT_ERR_SUCCESS$INT then

            //Create Log: DataMap Successfully Requested Publish for ...
            tmpPara1 := to_dint(pEntry^.iMid);
            tmpPara2 := pEntry^.pData$DINT;

            Logging_InterfLog(usLevel     :=  MQTTCLIENTINTERFACE_LOGGING_LEVEL_DEBUG,
                              dMsgGroup   :=  MQCLIINF_LOG_INFO_DATAMAP_ENTRY_PUBLISHED_GRP,
                              dMsgNbr     :=  MQCLIINF_LOG_INFO_DATAMAP_ENTRY_PUBLISHED_MSG,
                              pMsg        :=  MQCLIINF_LOG_INFO_DATAMAP_ENTRY_PUBLISHED_TEXT,
                              pPara1      :=  #tmpPara1,
                              pPara2      :=  #tmpPara2,
                              pPara3      :=  NIL,
                              pPara4      :=  NIL);

            pEntry^.State := DMPS_WaitForPublish;
            pEntry^.udLastAction := ops.tAbsolute;

          else

            //Create Log: DataMap Failed to issue Publish Request for ...

            tmpPara1 := to_dint(pEntry^.iMid);
            tmpPara2 := to_dint(iMQRet);

            Logging_InterfLog(usLevel     :=  MQTTCLIENTINTERFACE_LOGGING_LEVEL_ERR,
                              dMsgGroup   :=  MQCLIINF_LOG_ERROR_DATAMAP_PUBLISH_FAIL_MQCLI_GRP,
                              dMsgNbr     :=  MQCLIINF_LOG_ERROR_DATAMAP_PUBLISH_FAIL_MQCLI_MSG,
                              pMsg        :=  MQCLIINF_LOG_ERROR_DATAMAP_PUBLISH_FAIL_MQCLI_TEXT,
                              pPara1      :=  #tmpPara1,
                              pPara2      :=  #tmpPara2,
                              pPara3      :=  #pEntry^.pData$DINT,
                              pPara4      :=  NIL);

            pEntry^.State := DMPS_Error;

          end_if;

        //--------------------------------------------
        //Wait for feedback
        //--------------------------------------------
        t_e_DataMap_PublishStates::DMPS_WaitForPublish:

          //Wait For Feedback from the MQTT Client
          if pEntry^.bPublishComplete then

            //Create Log: Datamap, Publish Complete

            tmpPara1 := to_dint(pEntry^.iMid);
            tmpPara2 := pEntry^.pData$DINT;

            Logging_InterfLog(usLevel     :=  MQTTCLIENTINTERFACE_LOGGING_LEVEL_INFO,
                              dMsgGroup   :=  MQCLIINF_LOG_INFO_DATAMAP_ENTRY_PUB_COMP_GRP,
                              dMsgNbr     :=  MQCLIINF_LOG_INFO_DATAMAP_ENTRY_PUB_COMP_MSG,
                              pMsg        :=  MQCLIINF_LOG_INFO_DATAMAP_ENTRY_PUB_COMP_TEXT,
                              pPara1      :=  #tmpPara1,
                              pPara2      :=  #tmpPara2,
                              pPara3      :=  NIL,
                              pPara4      :=  NIL);

            pEntry^.bPublishComplete := FALSE;
            pEntry^.bInitialPublish := TRUE;
            pEntry^.State := DMPS_WaitForAction;

          end_if;

          //If the entry is moving on, free any temp mem associated with it.
          if pEntry^.State = DMPS_WaitForAction then

            //If this was a string
            if pEntry^.Datatype = DD_String then

              //If the entry had Tempmem associated with it, free it
              if pEntry^.pTempMem then

                MQTTClient.Free(mptr:=pEntry^.pTempMem);
                pEntry^.pTempMem := NIL;

              else

                tmpPara1 := to_dint(pEntry^.iMid);
                tmpPara2 := pEntry^.pData$DINT;

                Logging_InterfLog(usLevel     :=  MQTTCLIENTINTERFACE_LOGGING_LEVEL_WARNING,
                                  dMsgGroup   :=  MQCLIINF_LOG_WARNING_DATAMAP_PUBLISH_TMPPTR_NIL_GRP,
                                  dMsgNbr     :=  MQCLIINF_LOG_WARNING_DATAMAP_PUBLISH_TMPPTR_NIL_MSG,
                                  pMsg        :=  MQCLIINF_LOG_WARNING_DATAMAP_PUBLISH_TMPPTR_NIL_TEXT,
                                  pPara1      :=  #tmpPara1,
                                  pPara2      :=  #tmpPara2,
                                  pPara3      :=  NIL,
                                  pPara4      :=  NIL);
              end_if;

            end_if;

          end_if;

          //pEntry^.iMid := -1;

        //--------------------------------------------
        //Remove the Entry from the DataMap
        //--------------------------------------------
        t_e_DataMap_PublishStates::DMPS_Remove:

          //Remove this entry
          if udCount < (Config.pDataMapConfig^.udPublishElements - 1) then

            SigCLib.MemCpy( dst0  :=  pEntry,
                            src0  :=  (pEntry$UDINT + (sizeof(t_s_DataMap_ElementEntry_Publish)))$^void,
                            len0  :=  (sizeof(t_s_DataMap_ElementEntry_Publish))*(Config.pDataMapConfig^.udPublishElements - 1 - udCount));

          end_if;

          Config.pDataMapConfig^.udPublishElements -= 1;

          return;

        //--------------------------------------------
        //Error Occurred
        //--------------------------------------------
        t_e_DataMap_PublishStates::DMPS_Error:

          pEntry^.iMid := -1;
          //v1.13
          //In case an error occurs the topic should be recognized as not sent and will be sent as soon as the error is gone
          pEntry^.udCRC := 0;

          //If the reset time is set, wait for reset
          if (cDataMapResetTimeout <> 0) &
             (ops.tAbsolute - pEntry^.udLastAction >= cDataMapResetTimeout) then

            pEntry^.State := DMPS_Ready;

          end_if;

      end_case;

    end_for;

  end_if;

END_FUNCTION

FUNCTION MQTTClient_Interface::DataMap_ProcessMap_Subscribe
  VAR
  	pEntry : ^t_s_DataMap_ElementEntry_Subscribe;
    udCount : UDINT;
    iRetCode : INT;
    tmpPara1 : DINT;
    tmpPara2 : DINT;
  END_VAR

  //Process the Subscribe List
  if Config.pDataMapConfig^.udSubscribeElements > 0 then

    for udCount := 0 to Config.pDataMapConfig^.udSubscribeElements - 1 do

      pEntry$UDINT := ((Config.pDataMapConfig^.Elements.pSubscribeEntries)$UDINT + (udCount*sizeof(t_s_DataMap_ElementEntry_Subscribe)));

      //=========================================================
      //Entry FSM
      //=========================================================
      case pEntry^.State of

        //----------------------------------------------------
        //Ready to start operation, initialise
        //----------------------------------------------------
        t_e_DataMap_SubscribeStates::DMSS_Ready:

          //Reset Mid
          pEntry^.iMid  := -1;
          pEntry^.State := DMSS_Subscribe;

        //----------------------------------------------------
        //Issue Subscribe Request
        //----------------------------------------------------
        t_e_DataMap_SubscribeStates::DMSS_Subscribe:

          iRetCode := MQTT_Subscribe( pTopic      :=  #pEntry^.aTopic[0],
                                      iQoS        :=  pEntry^.iQos,
                                      pThis       :=  this,
                                      pCallback   :=  #DataMap_Return_Callback(),
                                      pMid        :=  #pEntry^.iMid,
                                      pApplMsgID  :=  #pEntry^.udApplMsgID);

          if iRetCode = MQTT_ERR_SUCCESS$INT then
            //Create Log: Subscribed DataMap Element, Element=XXXX

            tmpPara1 := to_dint(pEntry^.iMid);
            tmpPara2 := pEntry^.pData$DINT;

            Logging_InterfLog(usLevel     :=  MQTTCLIENTINTERFACE_LOGGING_LEVEL_DEBUG,
                              dMsgGroup   :=  MQCLIINF_LOG_INFO_DATAMAP_ENTRY_SUBD_GRP,
                              dMsgNbr     :=  MQCLIINF_LOG_INFO_DATAMAP_ENTRY_SUBD_MSG,
                              pMsg        :=  MQCLIINF_LOG_INFO_DATAMAP_ENTRY_SUBD_TEXT,
                              pPara1      :=  #tmpPara1,
                              pPara2      :=  NIL,
                              pPara3      :=  NIL,
                              pPara4      :=  NIL);

            pEntry^.State := DMSS_WaitForSubscribe;
            pEntry^.udLastAction := ops.tAbsolute;

          else
            //Create Log: Failed to Subscribe DataMap Element, MQTTClient Subscribe returned:XX, Element=XXXX

            tmpPara1 := to_dint(pEntry^.iMid);
            tmpPara2 := to_dint(iRetCode);

            Logging_InterfLog(usLevel     :=  MQTTCLIENTINTERFACE_LOGGING_LEVEL_ERR,
                              dMsgGroup   :=  MQCLIINF_LOG_ERROR_DATAMAP_SUBSCRIBE_FAIL_MQCLI_GRP,
                              dMsgNbr     :=  MQCLIINF_LOG_ERROR_DATAMAP_SUBSCRIBE_FAIL_MQCLI_MSG,
                              pMsg        :=  MQCLIINF_LOG_ERROR_DATAMAP_SUBSCRIBE_FAIL_MQCLI_TEXT,
                              pPara1      :=  #tmpPara1,
                              pPara2      :=  #tmpPara2,
                              pPara3      :=  #pEntry^.pData$DINT,
                              pPara4      :=  NIL);

            pEntry^.State := DMSS_Error;
            pEntry^.udLastAction := ops.tAbsolute;

          end_if;

        //----------------------------------------------------
        //Wait for Subscribe confirmation
        //----------------------------------------------------
        t_e_DataMap_SubscribeStates::DMSS_WaitForSubscribe:

          if ops.tAbsolute - pEntry^.udLastAction >= cDataMapSubTimeout then

            //Create Log: DataMap Failed to subscribe Entry, Timeout. retry.

            tmpPara1 := to_dint(pEntry^.iMid);
            tmpPara2 := pEntry^.pData$DINT;

            Logging_InterfLog(usLevel     :=  MQTTCLIENTINTERFACE_LOGGING_LEVEL_ERR,
                              dMsgGroup   :=  MQCLIINF_LOG_ERROR_DATAMAP_SUBSCRIBE_FAIL_TIMEOUT_GRP,
                              dMsgNbr     :=  MQCLIINF_LOG_ERROR_DATAMAP_SUBSCRIBE_FAIL_TIMEOUT_MSG,
                              pMsg        :=  MQCLIINF_LOG_ERROR_DATAMAP_SUBSCRIBE_FAIL_TIMEOUT_TEXT,
                              pPara1      :=  #tmpPara1,
                              pPara2      :=  #cDataMapSubTimeout$DINT,
                              pPara3      :=  #tmpPara2,
                              pPara4      :=  NIL);

            pEntry^.State := DMSS_Ready;

          end_if;

        //----------------------------------------------------
        //Subscribed
        //----------------------------------------------------
        t_e_DataMap_SubscribeStates::DMSS_Subscribed:

        //----------------------------------------------------
        //Issue Unsubscribe Command
        //----------------------------------------------------
        t_e_DataMap_SubscribeStates::DMSS_Unsubscribe:

          iRetCode := MQTT_Unsubscribe( pApplMsgID  :=  #pEntry^.udApplMsgID,
                                        pTopic      :=  NIL,
                                        pMid        :=  #pEntry^.iMid,
                                        pThis       :=  NIL,
                                        pCallback   :=  NIL);

          if iRetCode = MQTT_ERR_SUCCESS$INT then
            //Create Log: Subscribed DataMap Element, Element=XXXX

            tmpPara1 := to_dint(pEntry^.iMid);
            tmpPara2 := pEntry^.pData$DINT;

            Logging_InterfLog(usLevel     :=  MQTTCLIENTINTERFACE_LOGGING_LEVEL_DEBUG,
                              dMsgGroup   :=  MQCLIINF_LOG_INFO_DATAMAP_ENTRY_UNSUBD_GRP,
                              dMsgNbr     :=  MQCLIINF_LOG_INFO_DATAMAP_ENTRY_UNSUBD_MSG,
                              pMsg        :=  MQCLIINF_LOG_INFO_DATAMAP_ENTRY_UNSUBD_TEXT,
                              pPara1      :=  #tmpPara1,
                              pPara2      :=  #tmpPara2,
                              pPara3      :=  NIL,
                              pPara4      :=  NIL);

            //If this state has not already been changed by a phony callback (made from within MQTT_Unsubscribe), then change the state
            //to DMSS_WaitForUnsubscribe as we are actually still waiting for a callback.
            if pEntry^.State = DMSS_Unsubscribe then
              pEntry^.State := DMSS_WaitForUnsubscribe;
            end_if;

            pEntry^.udLastAction := ops.tAbsolute;

          elsif iRetCode = MQTTClient::MQTT_ERR_ALREADY_SUB$INT then

            // The Subscription was already there
            pEntry^.State := DMSS_Subscribed;
            pEntry^.udLastAction := ops.tAbsolute;

          else

            //Create Log: Failed to Subscribe DataMap Element, MQTTClient Subscribe returned:XX, Element=XXXX

            tmpPara1 := to_dint(pEntry^.iMid);
            tmpPara2 := to_dint(iRetCode);
